FUNCTION_BLOCK "Jdrk_RS_WS_N01_8"   // FB31, SCL
{ S7_Optimized_Access := 'TRUE' }
VERSION : 0.1
   VAR_OUTPUT
      Temperature : Real;
   END_VAR
   VAR_IN_OUT
      mb_query : "mb_query";
   END_VAR
   VAR
      sb : "mb_station_block_udt";
   END_VAR
   VAR RETAIN
      offset : Real;
   END_VAR
   VAR_TEMP
      tmp : Int;
   END_VAR
BEGIN
   // JDRK - RS-WS-N01-8 - Temperature and Humidity sensor

   "mb_station_block_header"(sb := #sb, mb_query := #mb_query);

   #mb_query(mb_addr := 1,
             mode := #mb_query.c.read.input_reg,
             data_addr := 1,
             data_ptr := #tmp);

   IF #mb_query.Done THEN
       #Temperature := INT_TO_REAL(#tmp) / 10 + #offset;
   END_IF;

   "mb_station_block_footer"(sb := #sb, mb_query := #mb_query);
END_FUNCTION_BLOCK

FUNCTION_BLOCK "keller_pressure_transmitters"   // FB32, SCL
{ S7_Optimized_Access := 'TRUE' }
VERSION : 0.1
   VAR_INPUT
      mb_addr : USInt;
   END_VAR
   VAR_IN_OUT
      mb_query : "mb_query";
   END_VAR
   VAR
      sb : "mb_station_block_udt";
      data : Struct
         pressure_sensor_1 : Real;
         pressure_sensor_2 : Real;
         temperature : Real;
         temperature_sensor_1 : Real;
         temperature_sensor_2 : Real;
      END_STRUCT;
   END_VAR
BEGIN
   // Keller, Series 30 and Series 40 - Pressure transmitters
   // 
   // http://www.keller-druck.com/picts/pdf/engl/comm_protocol_e.pdf

   "mb_station_block_header"(sb := #sb,
                             mb_query := #mb_query);

   #mb_query(mb_addr := #mb_addr,
             mode := #mb_query.c.read.holding_reg,
             data_addr := 2,
             data_ptr := #data);

   "mb_station_block_footer"(sb := #sb,
                             mb_query := #mb_query);
END_FUNCTION_BLOCK

FUNCTION_BLOCK "Mjk_expert"   // FB35, SCL
{ S7_Optimized_Access := 'TRUE' }
VERSION : 0.1
   VAR_INPUT
      mb_addr : USInt;
   END_VAR
   VAR_IN_OUT
      mb_query : "mb_query";
   END_VAR
   VAR
      sb : "mb_station_block_udt";
      data : Struct
         CH0 : Real;   // calculated_value (User-specific)
         P1 : Real;   // Pressure sensor 1
         P2 : Real;   // Pressure sensor 2
         T : Real;   // Temperature
         T1 : Real;   // Temperature sensor 1
         T2 : Real;   // Temperature sensor 2
      END_STRUCT;
   END_VAR
BEGIN
   // MJK - Expert 700-7060-7070 - Pressure transmitters

   "mb_station_block_header"(sb := #sb,
                             mb_query := #mb_query);
   #mb_query.mb_addr := #mb_addr;

   #mb_query.mode := #mb_query.c.read.holding_reg;
   #mb_query(data_addr := 0,
             data_ptr := #data);

   "mb_station_block_footer"(sb := #sb,
                             mb_query := #mb_query);
END_FUNCTION_BLOCK

FUNCTION_BLOCK "Moxa_ioLogik_R1200"   // FB36, SCL
{ S7_Optimized_Access := 'TRUE' }
VERSION : 0.1
   VAR_INPUT
      mb_addr : UInt;
   END_VAR
   VAR_IN_OUT
      mb_query : "mb_query";
   END_VAR
   VAR
      sb : "mb_station_block_udt";
      in : Array[0..15] of Bool;
      out : Array[0..15] of Bool;
   END_VAR
BEGIN
   // Moxa - ioLogik R1200
   // 
   // Web: https://www.moxa.com/doc/man/ioLogik_R1200_Series_UM_e3.1.pdf

   "mb_station_block_header"(sb := #sb,
                             mb_query := #mb_query);
   #mb_query.mb_addr := #mb_addr;

   #mb_query(mode := #mb_query.c.read.discrete_input,
             data_addr := 0,
             data_ptr := #in);

   #mb_query(mode := #mb_query.c.write.discrete_output,
             data_addr := 16#140,
             data_ptr := #out);

   "mb_station_block_footer"(sb := #sb,
                             mb_query := #mb_query);
END_FUNCTION_BLOCK

FUNCTION_BLOCK "MTS_sensors_M_Series"   // FB37, SCL
{ S7_Optimized_Access := 'TRUE' }
VERSION : 0.1
   VAR_INPUT
      mb_addr : UInt;
   END_VAR
   VAR_OUTPUT
      level : Real;
      temperature : Real;
   END_VAR
   VAR_IN_OUT
      mb_query : "mb_query";
   END_VAR
   VAR
      sb : "mb_station_block_udt";
      query_1 : Struct
         product_level : DInt;
         Interface_level : DInt;
         roof_level : DInt;
         temperature : Array[1..5] of DInt;
         temperature_avg : DInt;
      END_STRUCT;
   END_VAR
BEGIN
   // MTS sensors - M-Series - Liquid-Level Sensors
   // Web: http://www.mtssensors.com/fileadmin/media/pdfs/550791.pdf

   "mb_station_block_header"(sb := #sb,
                             mb_query := #mb_query);
   #mb_query.mb_addr := #mb_addr;

   #mb_query.mode := #mb_query.c.mode.read;
   #mb_query(data_addr := 30001,
             data_ptr := #query_1);

   "mb_station_block_footer"(sb := #sb,
                             mb_query := #mb_query);

   #level := DINT_TO_REAL(#query_1.product_level) * 0.001;
   #temperature := DINT_TO_REAL(#query_1.temperature_avg) * 0.0001;
END_FUNCTION_BLOCK

FUNCTION_BLOCK "Novus_tht"   // FB38, SCL
{ S7_Optimized_Access := 'TRUE' }
VERSION : 0.1
   VAR_INPUT
      mb_addr : USInt;
   END_VAR
   VAR_OUTPUT
      temperature : Int;
      humidity : Int;
   END_VAR
   VAR_IN_OUT
      mb_query : "mb_query";
   END_VAR
   VAR
      sb : "mb_station_block_udt";
      serial_number : DWord;
      raw_values : Struct
         temp : Int;
         hum : Int;
      END_STRUCT;
   END_VAR
BEGIN
   // - Novus - RHT (Temperature transmitter)
   // - http://www.novusautomation.com/downloads/Arquivos/v10x_b_manual_rht_wm-dm-p10_485_lcd_%20english.pdf

   "mb_station_block_header"(sb := #sb, mb_query := #mb_query);
   #mb_query.mb_addr := #mb_addr;

   #mb_query.mode := #mb_query.c.read.holding_reg;
   #mb_query(data_addr := 7, data_ptr := #raw_values);
   #mb_query(data_addr := 0, data_ptr := #serial_number);

   "mb_station_block_footer"(sb := #sb, mb_query := #mb_query);

   #temperature := #raw_values.temp / 10;
   #humidity := #raw_values.hum / 10;
END_FUNCTION_BLOCK

FUNCTION_BLOCK "Onicon_F5100"   // FB39, SCL
{ S7_Optimized_Access := 'TRUE' }
VERSION : 0.1
   VAR_INPUT
      mb_addr : USInt;
   END_VAR
   VAR_IN_OUT
      mb_query : "mb_query";
   END_VAR
   VAR
      sb : "mb_station_block_udt";
      reset : Bool;
      query1 : Struct
         flow_total : UDInt;
      END_STRUCT;
      query2 : Struct
         flow_rate : Real;
         temperature : Real;
      END_STRUCT;
   END_VAR
BEGIN
   // Onicon - F-5100
   // http://www.onicon.com/pdfs/0669-7-F-5100-MOD-Network-Interface-Installation-Guide-09-15.pdf

   "mb_station_block_header"(sb := #sb,
                             mb_query := #mb_query);
   #mb_query.mb_addr := #mb_addr;

   #mb_query.data_addr := 312; // 313 - 1
   IF #reset THEN
       #query1.flow_total := 0;
       #mb_query(mode := #mb_query.c.write.holding_reg,
                 data_ptr := #query1.flow_total);
       IF #mb_query.stat.done THEN
           #reset := false;
       END_IF;
   ELSE
       #mb_query(mode := #mb_query.c.read.holding_reg,
                 data_ptr := #query1);
   END_IF;

   #mb_query(mode := #mb_query.c.read.holding_reg,
             data_addr := 578, // 579 - 1,
             data_ptr := #query2);

   "mb_station_block_footer"(sb := #sb,
                             mb_query := #mb_query);
END_FUNCTION_BLOCK

FUNCTION_BLOCK "Phoenix_Contact_UPS"   // FB40, SCL
{ S7_Optimized_Access := 'TRUE' }
VERSION : 0.1
   VAR_INPUT
      mb_addr : UInt;
   END_VAR
   VAR_IN_OUT
      mb_query : "mb_query";
   END_VAR
   VAR
      sb : "mb_station_block_udt";
      read1 : Struct
         remote : Word;
         BatteryMode : Word;
         ShutdownEvent : Word;
         BatteryCharging : Word;
      END_STRUCT;
      read2 : Struct
         OutputVoltage_mV : UInt;
      END_STRUCT;
      read3 : Struct
         SocStateOfCharge : UInt;   // [%]
         SocResidualBackupTimeM : UInt;   // Minute
      END_STRUCT;
      read4 : Struct
         BatteryVoltage_mV : UInt;
         BatteryTemperature : UInt;   // Kelvin
         OutputVoltage2_mV : UInt;
         SocResidualBackupTimeS : UInt;
         BatteryNomCapacityWs : UInt;
      END_STRUCT;
      read5 : Struct
         BatteryDischaCurrent : UInt;
         BatteryDetectedUnits : UInt;
         BatteryNomCapacitymAh : UInt;
         BatteryInstalledType : UInt;
      END_STRUCT;
      read6_Alarm : Struct
         x08 : Bool;
         x09_no_battery : Bool;
         x10_inconsistent_technology : Bool;
         x11_overload_cutoff : Bool;
         "x12_Low_battery_(Voltage)" : Bool;
         "x13_Low_battery_(Charge)" : Bool;
         "x14_Low_battery_(Time)" : Bool;
         x15 : Bool;
         "x00_End_of_life_(SOH)" : Bool;
         x01 : Bool;
         x02 : Bool;
         x03 : Bool;
         "x04_End_of_life_(Resitance)" : Bool;
         "x05_Endof_life_(Resitance)" : Bool;
         "x06_End_of_life_(Time)" : Bool;
         "x07_End_of_life_(Voltage)" : Bool;
      END_STRUCT;
   END_VAR
BEGIN
   // Phoenix Contact - UPS
   // QUINT UPS-IQ, TRIO-UPS
   // Web: https://media.digikey.com/pdf/Data%20Sheets/
   //      Phoenix%20Contact%20PDFs/2320461_Ds.pdf

   "mb_station_block_header"(sb := #sb, mb_query := #mb_query);
   #mb_query.mb_addr := #mb_addr;

   #mb_query.mode := #mb_query.c.read.holding_reg;
   #mb_query(data_addr := 29696, data_ptr := #read1);
   #mb_query(data_addr := 29745, data_ptr := #read2);
   #mb_query(data_addr := 29749, data_ptr := #read3);
   #mb_query(data_addr := 29792, data_ptr := #read4);
   #mb_query(data_addr := 29798, data_ptr := #read5);
   #mb_query(data_addr := 29840, data_ptr := #read6_Alarm);

   "mb_station_block_footer"(sb := #sb, mb_query := #mb_query);
END_FUNCTION_BLOCK

FUNCTION_BLOCK "Rotork_Mk_3_option_card"   // FB44, SCL
{ S7_Optimized_Access := 'TRUE' }
VERSION : 0.1
   VAR_INPUT
      mb_addr : UInt;
   END_VAR
   VAR_IN_OUT
      mb_query : "mb_query";
   END_VAR
   VAR
      sb : "mb_station_block_udt";
      read1 : Struct
         x00_actuator_moving : Bool;
         "x01_Close position limit" : Bool;
         "x02_Open position limit" : Bool;
         "x03_Valve running close" : Bool;
         "x04_Valve running open" : Bool;
         "x05_Selector in remote" : Bool;
         "x06_Selector in local stop" : Bool;
         "x07_Selector in local" : Bool;
         "x08_Thermostat tripped" : Bool;
         "x09_Monitor relay" : Bool;
         "x10_Valve obstructed" : Bool;
         "x11_Valve jammed" : Bool;
         "x12_Manual movement" : Bool;
         "x13_MIT_Interrupter timer" : Bool;
         "x14_Position control enabled" : Bool;
         "x15_Watchdog Recovery" : Bool;
         "x16_Battery low" : Bool;
         "x17_Open Interlock input active" : Bool;
         "x18_Close Interlock input active" : Bool;
         "x19_Hard wired input DI-1 (open)" : Bool;
         "x20_Hard wired input DI-2 (close)" : Bool;
         "x21_Hard wired input DI-3 (stop)" : Bool;
         "x22_Hard wired input DI-4 (ESD)" : Bool;
         x23 : Bool;
         x24 : Bool;
         x25 : Bool;
         "x26_Control contention" : Bool;
         "x27_Partial stroke test in progress" : Bool;
         "x28_Partial stroke test error" : Bool;
         "x29_General alarm" : Bool;
         x30 : Bool;
         x31 : Bool;
      END_STRUCT;
      read2 : Struct
         instantaneous_torque : Int;
         valve_position : Int;   // x10 %
         analogue_input : Int;
      END_STRUCT;
      write1 : Struct
         stop : Bool;
         close : Bool;
         open : Bool;
         emergency_shut_down : Bool;
         output_DO_1 : Bool;
         output_DO_2 : Bool;
         output_DO_3 : Bool;
         output_DO_4 : Bool;
      END_STRUCT;
      write2 : Struct
         actuator_digital_control : Bool;
         position_demand_output : Bool;
      END_STRUCT;
      actuator_tag_name : String[12];
      action_on_loss_of_comms : Int;
   END_VAR
BEGIN
   // Rotork  - Mk 3 Option Card

   // http://www.rotork.com/en/product/index/modbusliterature
   // Publication PUB091-004-00_0715

   "mb_station_block_header"(sb := #sb, mb_query := #mb_query);
   #mb_query.mb_addr := #mb_addr;

   #mb_query.mode := #mb_query.c.read.discrete_input;
   #mb_query(data_addr := 0, data_ptr := #read1);

   #mb_query.mode := #mb_query.c.read.holding_reg;
   #mb_query(data_addr := 2, data_ptr := #read2);
   #mb_query(data_addr := 26, data_ptr := #actuator_tag_name);

   #mb_query.mode := #mb_query.c.write.discrete_output;
   #mb_query(data_addr := 0, data_ptr := #write1);

   #mb_query.mode := #mb_query.c.write.holding_reg;
   // 0=No-Action, 1=Open, 3=Close, 5=Stop, 7=Position
   #mb_query(data_addr := 7, data_ptr := #action_on_loss_of_comms);
   #mb_query(data_addr := 5, data_ptr := #write2);

   "mb_station_block_footer"(sb := #sb, mb_query := #mb_query);
END_FUNCTION_BLOCK

FUNCTION_BLOCK "SensorsONE_DCT_531"   // FB52, SCL
{ S7_Optimized_Access := 'TRUE' }
VERSION : 0.1
   VAR_INPUT
      mb_addr : UInt;
   END_VAR
   VAR_IN_OUT
      mb_query : "mb_query";
   END_VAR
   VAR
      sb : "mb_station_block_udt";
      data : Struct
         serial_number : UDInt;
         date_last_calibration : UDInt;
         upper_range_pressure : Real;
         lower_range_pressure : Real;
         actual_pressure : Real;
         max_pressure : Real;
         min_pressure : Real;
         upper_range_temperature : Real;
         lower_range_temperature : Real;
         actual_temperature : Real;
         max_temperature : Real;
         min_temperature : Real;
      END_STRUCT;
   END_VAR
BEGIN
   // SensorsONE - DCT 531
   // 
   // https://www.sensorsone.com/dct-531-modbus-rtu-rs485-pressure-sensor/

   "mb_station_block_header"(sb := #sb,
                             mb_query := #mb_query);
   #mb_query.mb_addr := #mb_addr;

   #mb_query.mode := #mb_query.c.read.input_reg;
   #mb_query(data_addr := 0,
             data_ptr := #data);

   "mb_station_block_footer"(sb := #sb,
                             mb_query := #mb_query);
END_FUNCTION_BLOCK

FUNCTION_BLOCK "Sierra_thermal_mass_flow_meters"   // FB61, SCL
{ S7_Optimized_Access := 'TRUE' }
VERSION : 0.1
   VAR_INPUT
      mb_addr : UInt;
      reset_totalizer : Bool := 1;
   END_VAR
   VAR_IN_OUT
      mb_query : "mb_query";
   END_VAR
   VAR
      sb : "mb_station_block_udt";
      data : Struct
         flow : Real;
         totalizer : DInt;
      END_STRUCT;
      serial_number : String[12];
   END_VAR
   VAR_TEMP
      "int" : Int;
   END_VAR
BEGIN
   // Sierra - 600/700 Series - Thermal mass flow meters
   // Models: 620S, 620S-BT, 640S, 760S, 780S, and 780S-UHP

   // Web: https://www.ccontrols.com/support/dp/600-700-modbus-instruction-manual.pdf

   "mb_station_block_header"(sb := #sb,
                             mb_query := #mb_query);
   #mb_query.mb_addr := #mb_addr;

   #mb_query.mode := #mb_query.c.mode.read;
   #mb_query(data_addr := 40001,
             data_ptr := #data);
   #mb_query(data_addr := 40016,
             data_ptr := #serial_number);

   IF #reset_totalizer THEN
       #mb_query.mode := #mb_query.c.mode.write;
       #"int" := 1;
       #mb_query(data_addr := 40008,
                 data_ptr := #"int");
   END_IF;

   "mb_station_block_footer"(sb := #sb,
                             mb_query := #mb_query);
END_FUNCTION_BLOCK

FUNCTION_BLOCK "Smart_biene_sb_hl"   // FB62, SCL
{ S7_Optimized_Access := 'TRUE' }
VERSION : 0.1
   VAR_INPUT
      mb_addr : UInt;
   END_VAR
   VAR_IN_OUT
      mb_query : "mb_query";
   END_VAR
   VAR
      s : "mb_station_block_udt";
      data : Struct
         "Min measuring range" : Word;
         "Max measuring range" : Word;
         "Pressure Value" : Word;
         "High Pressure" : Word;
         "Low Pressure" : Word;
         stat : Word;
         model : String[12];
         serial : String[12];
         unit : Int;
      END_STRUCT;
      "a" : Struct
         x08 : Bool;
         x09 : Bool;
         x10 : Bool;
         x11 : Bool;
         x12 : Bool;
         x13 : Bool;
         x14 : Bool;
         x15 : Bool;
         x00 : Bool;
         x01 : Bool;
         x02 : Bool;
         x03 : Bool;
         x04 : Bool;
         x05 : Bool;
         x06 : Bool;
         x07 : Bool;
      END_STRUCT;
   END_VAR
BEGIN
   // Smart Biene - SB-HL - Hydrostatic Level Transmitter
   // 
   // Web: http://smartbiene.com/images/pdf/hydrostatic-level/
   //      Hydrostatic%20level-SP-HL-01-ModbusRTU.pdf

   "mb_station_block_header"(sb := #s,
                             mb_query := #mb_query);
   #mb_query.mb_addr := #mb_addr;

   #mb_query.mode := #mb_query.c.read.holding_reg;
   #mb_query(data_addr := 0,
             data_ptr := #data);

   "mb_station_block_footer"(sb := #s,
                             mb_query := #mb_query);

   (*
   Unit:
   0-mbar
   1-bar
   2-PSI
   3-KPa
   4-MPa
   5-Kg/cm2
   6-mmHg
   7-mmH2O
   8-inHg
   9-inH2O 
   *)
END_FUNCTION_BLOCK

FUNCTION_BLOCK "Socomec_diris"   // FB63, SCL
{ S7_Optimized_Access := 'TRUE' }
VERSION : 0.1
   VAR_INPUT
      mb_addr : USInt;
      old_mapping : Bool;
   END_VAR
   VAR_OUTPUT
      data : Struct
         voltage_L_L : Array[1..3] of Real;   // 1->L1-L2, 2->L2-L3, 3->L3-L1
         voltage_L_N : Array[1..3] of Real;
         frequency : Real;
         current : Array[1..3] of Real;
         neutral_current : Real;
         sum_active_power : Real;
         sum_reactive_power : Real;
         sum_apparent_power : Real;
         sum_power_factor : Real;   // -: leading and + : lagging
         power_active : Array[1..3] of Real;
         power_reactive : Array[1..3] of Real;
         power_apparent : Array[1..3] of Real;
         power_factor : Array[1..3] of Real;
      END_STRUCT;
   END_VAR
   VAR_IN_OUT
      mb_query : "mb_query";
   END_VAR
   VAR
      sb : "mb_station_block_udt";
      query_1 : Struct
         voltage_L_L : Array[1..3] of DInt;   // 1->L1-L2, 2->L2-L3, 3->L3-L1
         voltage_L_N : Array[1..3] of DInt;
         frequency : DInt;
         current : Array[1..3] of DInt;
         neutral_current : DInt;
         sum_active_power : DInt;
         sum_reactive_power : DInt;
         sum_apparent_power : DInt;
         sum_power_factor : DInt;   // -: leading and + : lagging
         power_active : Array[1..3] of DInt;
         power_reactive : Array[1..3] of DInt;
         power_apparent : Array[1..3] of DInt;
         power_factor : Array[1..3] of DInt;
      END_STRUCT;
      query_2_temperature : DInt;
   END_VAR
   VAR_TEMP
      j : Int;
   END_VAR
BEGIN
   // Socomec Diris A40/A41 - Power meter
   // https://www.socomec.com/files/live/sites/systemsite/files/SCP/
   // 6_gestion_energie/diris/diris_a40/536181B_GB_Ethernet.pdf

   // old_mapping:
   // http://www.ferrazshawmutsales.com/pdfs/cdr_27038_RS485_JBus-ModBus.pdf

   "mb_station_block_header"(sb := #sb,
                             mb_query := #mb_query);
   #mb_query.mb_addr := #mb_addr;

   #mb_query.mode := #mb_query.c.read.holding_reg;

   #mb_query(data_addr := SEL(G := #old_mapping, IN0 := 50514, IN1 := 768),
             data_ptr := #query_1);

   IF NOT #old_mapping THEN
       #mb_query(data_addr := 51457,
                 data_ptr := #query_2_temperature);
   END_IF;

   "mb_station_block_footer"(sb := #sb,
                             mb_query := #mb_query);

   (* IF #s.out.error_comm THEN
       FOR #j := 1 TO 3 DO
           #query_1.voltage_L_L[#j] := 0;
           #query_1.voltage_L_N[#j] := 0;
           #query_1.current[#j] := 0;
           #query_1.power_active[#j] := 0;
           #query_1.power_reactive[#j] := 0;
           #query_1.power_apparent[#j] := 0;
           #query_1.power_factor[#j] := 0;
       END_FOR;
       #query_1.frequency := 0;
       #query_1.neutral_current := 0;
       #query_1.sum_active_power := 0;
       #query_1.sum_reactive_power := 0;
       #query_1.sum_apparent_power := 0;
       #query_1.sum_power_factor := 0;

       #query_2_temperature := 0;
   END_IF; // *)

   FOR #j := 1 TO 3 DO
       #data.voltage_L_L[#j] := DINT_TO_REAL(#query_1.voltage_L_L[#j]) / 100;
       #data.voltage_L_N[#j] := DINT_TO_REAL(#query_1.voltage_L_N[#j]) / 100;
       #data.current[#j] := DINT_TO_REAL(#query_1.current[#j]) / 1000;
       #data.power_active[#j] := DINT_TO_REAL(#query_1.power_active[#j]) / 100;
       #data.power_reactive[#j] := DINT_TO_REAL(#query_1.power_reactive[#j]) / 100;
       #data.power_apparent[#j] := DINT_TO_REAL(#query_1.power_apparent[#j]) / 100;
       #data.power_factor[#j] := DINT_TO_REAL(#query_1.power_factor[#j]) / 1000;
   END_FOR;
   #data.frequency := DINT_TO_REAL(#query_1.frequency) / 100;
   #data.neutral_current := DINT_TO_REAL(#query_1.neutral_current) / 100;
   #data.sum_active_power := DINT_TO_REAL(#query_1.sum_active_power) / 100;
   #data.sum_reactive_power := DINT_TO_REAL(#query_1.sum_reactive_power) / 100;
   #data.sum_apparent_power := DINT_TO_REAL(#query_1.sum_apparent_power) / 100;
   #data.sum_power_factor := DINT_TO_REAL(#query_1.sum_power_factor) / 1000;
END_FUNCTION_BLOCK

FUNCTION_BLOCK "Sparling_Instruments_Tiger_Mag"   // FB64, SCL
{ S7_Optimized_Access := 'TRUE' }
VERSION : 0.1
   VAR_INPUT
      mb_addr : USInt;
   END_VAR
   VAR_IN_OUT
      mb_query : "mb_query";
   END_VAR
   VAR
      sb : "mb_station_block_udt";
      read1 : Struct
         flow : Real;   // 0.01 [Hz]
         total_fwd : UDInt;   // 0.1 [A]
         total_rev : UDInt;
         unit_flow : String[4];
         unit_total : String[4];
         total_registration : Real;
      END_STRUCT;
      serial_number : UDInt;
   END_VAR
BEGIN
   // Sparling Instruments - Tiger Mag 
   // FM656, FM657, FM626, FM627, FM626 Sanitary
   // http://www.sparlinginstruments.com/documents/IDS-TMEP-160323.PDF
   // Revision 160323

   "mb_station_block_header"(sb := #sb,
                             mb_query := #mb_query);
   #mb_query.mb_addr := #mb_addr;

   #mb_query.mode := #mb_query.c.mode.read;
   #mb_query(data_addr := 30001,
             data_ptr := #read1);
   #mb_query(data_addr := 31003,
             data_ptr := #serial_number);

   "mb_station_block_footer"(sb := #sb,
                             mb_query := #mb_query);

   (*
   Terminal RS-485 Bus:
   1-RX  -> A+
   2-TX  -> B-
   3-GND -> GND
   4-DTR -> N/A Not used

   Default comm. param:
   19200 bps, even parity. 
    Slave ID: 1.
   *)
END_FUNCTION_BLOCK

FUNCTION_BLOCK "Syxthsense_TEHR_M"   // FB70, SCL
TITLE = Syxthsense - TEHR-M - Temperature transmitter
{ S7_Optimized_Access := 'TRUE' }
AUTHOR : OlaBjornli
VERSION : 0.1
   VAR_INPUT
      mb_addr : USInt := 1;
   END_VAR
   VAR_OUTPUT
      temperature : Real;   // [Â°C]
      analogue_output : Real;   // [Â°F]
      potentiometer_position : Real;   // [%]
   END_VAR
   VAR_IN_OUT
      mb_query : "mb_query";
   END_VAR
   VAR
      sb : "mb_station_block_udt";
      read1 : Struct
         temperature : Int;   // [Â°C]
         analogue_output : Int;   // [Â°F]
         potentiometer_position : Int;   // [%]
      END_STRUCT;
   END_VAR
BEGIN
   // http://www.syxthsense.com/product/product_pdf/SN1.174-TEHR-M.pdf

   "mb_station_block_header"(sb := #sb, mb_query := #mb_query);

   #mb_query(mb_addr := #mb_addr,
             mode := #mb_query.c.mode.read,
             data_addr := 30001,
             data_ptr := #read1);
   #temperature := INT_TO_REAL(#read1.temperature) / 10;
   #analogue_output := INT_TO_REAL(#read1.analogue_output) / 10;
   #potentiometer_position := INT_TO_REAL(#read1.potentiometer_position) / 10;

   "mb_station_block_footer"(sb := #sb, mb_query := #mb_query);
END_FUNCTION_BLOCK

FUNCTION_BLOCK "Telemecanique_Schneider_Altivar_21_inverter"   // FB71, SCL
{ S7_Optimized_Access := 'TRUE' }
VERSION : 0.1
   VAR_INPUT
      mb_addr : UInt;
      ref : Real;
   END_VAR
   VAR_IN_OUT
      mb_query : "mb_query";
   END_VAR
   VAR
      sb : "mb_station_block_udt";
      read1 : Struct
         "Output frequency" : Word;
         stat : Struct
            x08 : Bool;
            x09_Reverse : Bool;
            x10_Run : Bool;
            x11_Coast_stop : Bool;
            x12_Emergency_stop : Bool;
            x13_Standby_ST_ON : Bool;   // Standby: Initialization completed, not failure stop status, not alarm stop status (MOFF, LL forced stop or forced stop due to a momentary power failure), ST=ON, and RUN=ON
            x14_Standby : Bool;   // Standby: Initialization completed, not failure stop status, and not alarm stop status (MOFF, LL forced stop or forced stop due to a momentary power failure)
            x15_Local : Bool;
            x00_Failure_FL : Bool;
            x01_Failure : Bool;
            x02_Alarm : Bool;
            x03_Main_circuit_undervoltage : Bool;
            x04_THR_2 : Bool;   // THR1: PT=set value, vL, vb, Thr - THR2: PT=0, F170, F172, F173
            x05_PI_control_OFF : Bool;
            x06_Acceleration2_deceleration2 : Bool;
            x07_DC_braking : Bool;
         END_STRUCT;
      END_STRUCT;
      read2 : Struct
         Command_mode : Int;   // 0:Terminal board, 1:Operation panel, 2:Serial
         "Setpoint mode" : Int;   // 1 VIA, 2 VIB, 3 Operation panel, 4 Serial, 5 TB up down frequency, 255 Preset speed operation
      END_STRUCT;
      read3_alarm : Struct
         x08_Over_torque : Bool;
         x09_Cumulative_operation_hours : Bool;
         x10 : Bool;
         x11 : Bool;
         x12 : Bool;
         "x13_Main circuit_undervoltage" : Bool;   // same as MS-relay status
         x14_Decelerating_stopping : Bool;   // Related: F256 setting. At the time of the instant blackout, Forced deceleration/stop
         x15_Decelerating_stopping : Bool;   // Related: F302 setting. An automatic stop during the lower limit frequency continuance
         x00_Overcurrent : Bool;
         x01_Inverter_overload : Bool;
         x02_Motor_overload : Bool;
         x03_Overheat : Bool;
         x04_Overvoltage : Bool;
         x05_Main_circuit_undervoltage : Bool;
         x06 : Bool;
         x07_Undercurrent : Bool;
      END_STRUCT;
      read4_alarm2 : Struct
         x08 : Bool;
         x09 : Bool;
         x10 : Bool;
         x11 : Bool;
         x12 : Bool;
         x13 : Bool;
         x14 : Bool;
         x15 : Bool;
         x00_Fan_life_alarm : Bool;
         x01_Circuit_board_life : Bool;
         x02_Main_circuit_capacitor_life : Bool;
         x03_User_set_alarm : Bool;
         x04 : Bool;
         x05 : Bool;
         x06 : Bool;
         x07 : Bool;
      END_STRUCT;
      read5_trip_code : UInt;
      write1 : Struct
         cmd : Struct
            x08 : Bool;
            x09_Reverse : Bool;
            x10_Run : Bool;
            x11_Coast_stop : Bool;
            x12_Emergency_stop : Bool;
            x13_Fault_reset : Bool;
            x14_Setpoint_priority : Bool;   // Enabled regardless of the setting of FMOD
            x15_Command_priority : Bool;   // Enabled regardless of the setting of CMOD
            x00_Preset_speed_b0 : Bool := TRUE;
            x01_Preset_speed_b1 : Bool;
            x02_Preset_speed_b2 : Bool;
            x03 : Bool;
            x04_thr2 : Bool;   // THR1 : PT=set value, vL, vb, tHr - THR2 : PT=0, F170, F172, F173
            x05_PI_control : Bool;   // 0:Normal operation, 1:PI OFF
            x06_Acceleration_deceleration_pattern_2 : Bool;   // 0: Acceleration deceleration pattern 1
            x07_DC_braking : Bool;
         END_STRUCT;
         ref : UInt;
      END_STRUCT;
   END_VAR
BEGIN
   // Telemecanique (Schneider) - Altivar 21 inverter
   // VFD (AC-drive)
   // http://www2.schneider-electric.com/resources/sites/SCHNEIDER_ELECTRIC/
   // content/live/FAQS/12000/FA12122/en_US/Altivar%2021%20Modbus%20manual.pdf

   "mb_station_block_header"(sb := #sb, mb_query := #mb_query);
   #mb_query.mb_addr := #mb_addr;

   #mb_query.mode := #mb_query.c.read.holding_reg;
   #mb_query(data_addr := 16#fd00, data_ptr := #read1);
   #mb_query(data_addr := 16#fe45, data_ptr := #read2);
   #mb_query(data_addr := 16#fe91, data_ptr := #read3_alarm);
   #mb_query(data_addr := 16#fe79, data_ptr := #read4_alarm2);
   #mb_query(data_addr := 16#FC90, data_ptr := #read5_trip_code);

   #write1.ref := REAL_TO_UINT(#ref * 100);
   #write1.cmd.x10_Run := #ref <> 0;
   #mb_query.mode := #mb_query.c.write.holding_reg;
   #mb_query(data_addr := 16#fa00, data_ptr := #write1);

   "mb_station_block_footer"(sb := #sb, mb_query := #mb_query);

   (* Trip code
   NErr     0  0  No error
   OC1      1  1  Over-current during acceleration
   OC2      2  2  Over-current during deceleration
   OC3      3  3  Over-current during constant speed operation
   OCL      4  4  Over-current in load at startup
   OCA      5  5  Short circuit in arm
   EPHI     8  8  Input phase failure
   EPHO     9  9  Output phase failure
   OP1      A 10 Overvoltage during acceleration
   OP2      B 11 Overvoltage during deceleration
   OP3      C 12 Overvoltage during constant speed operation
   OL1      D 13 Over-LOAD in inverter
   OL2      E 14 Over-LOAD in motor
   OH      10 16 Overheat trip
   E       11 17 Emergency stop
   EEP1    12 18 EEPROM fault 1 (writing error)
   EEP2    13 19 EEPROM fault 2 (reading error)
   EEP3    14 20 EEPROM fault 3 (internal fault)
   Err2    15 21 RAM fault
   Err3    16 22 ROM fault
   Err4    17 23 CPU fault
   Err5    18 24 Communication error trip
   Err7    1A 26 Current detector fault
   Err8    1B 27 Optional circuit board type error
   UC      1D 29 Small-current trip
   UP1     1E 30 Trip due to undervoltage in main circuit
   Ot      20 32 Over-torque trip
   EF2     22 34 Ground fault trip (hardware detection)
   OC1P    25 37 Overcurrent flowing in element during acceleration
   OC2P    26 38 Overcurrent flowing in element during deceleration
   OC3P    27 39 Overcurrent flowing in element during operation
   EtYP    29 41 Inverter type error
   OH2     2E 46 External thermal input
   SOUt    2F 47 VIA cable break
   E-18    32 50 Break in an analog signal cable
   E-19    33 51 CPU fault
   E-20    34 52 Excess torque boost
   E-21    35 53 CPU fault
   Etn1    54 84 Auto-tuning error
   *)
END_FUNCTION_BLOCK

FUNCTION_BLOCK "Vacon_OPTC2_C8"   // FB72, SCL
{ S7_Optimized_Access := 'TRUE' }
VERSION : 0.1
   VAR_INPUT
      mb_addr : UInt;
      ref : Real;
   END_VAR
   VAR_OUTPUT
      actual_speed : Real;
      Output_Frequency : Real;   // hz
      Motor_Speed : Real;   // rpm
      Motor_Current : Real;   // A
      Motor_Torque : Real;   // %
      Motor_Power : Real;   // %
      Motor_Voltage : Real;   // V
      DC_link_voltage : Real;   // V
   END_VAR
   VAR_IN_OUT
      mb_query : "mb_query";
   END_VAR
   VAR
      sb : "mb_station_block_udt";
      write : Struct
         ctw : Struct
            byte0 : Bool;
            x00_run : Bool;
            x01_reverse : Bool;
            x02_reset : Bool;
            x03 : Bool;
            x04 : Bool;
            x05 : Bool;
            x06 : Bool;
            x07 : Bool;
         END_STRUCT;
         "General Control Word" : Word;
         speed_reference : Int;
      END_STRUCT;
      read : Struct
         status : Struct
            x08_TC_Speed_Limit_Not_Active : Bool;
            x09_Detected_Encoder_Direction_Counterclockwise : Bool;
            x10_UV_Fast_Stop_Not_Active : Bool;
            x11 : Bool;
            x12 : Bool;
            x13 : Bool;
            x14 : Bool;
            x15 : Bool;
            x00_ready : Bool;
            x01_RUN : Bool;
            x02_reverse : Bool;
            x03_Faulted : Bool;
            x04_Warning : Bool;
            x05_Ref_Frequency_reached : Bool;
            x06_Motor_is_running_at_zero_speed : Bool;
            x07_Flux_Ready : Bool;
         END_STRUCT;
         general_status : Struct
            x08 : Bool;
            x09 : Bool;
            x10 : Bool;
            x11 : Bool;
            x12 : Bool;
            x13_Fieldbus_control : Bool;
            "x14_Panel control" : Bool;
            x15_IO_control : Bool;
            x00 : Bool;
            x01 : Bool;
            x02 : Bool;
            x03 : Bool;
            x04 : Bool;
            x05 : Bool;
            x06 : Bool;
            x07 : Bool;
         END_STRUCT;
         actual_speed : Int;
         Output_Frequency : Int;   // 0.01 Hz
         Motor_Speed : Int;   // 1 rpm
         Motor_Current : Int;   // 0.1 A
         Motor_Torque : Int;   // 0.1 %
         Motor_Power : Int;   // 0.1 %
         Motor_Voltage : Int;   // 0.1 V
         DC_link_voltage : Int;   // 1 V
         Active_Fault_Code : Int;
      END_STRUCT;
   END_VAR
BEGIN
   // Vacon NX - OPTC2/C8 - AC drives
   // Modbus/N2 option board
   // Document code: DPD00899A , Date 19.01.2012
   // Web: http://www.vacon.com/ImageVaultFiles/id_3118/cf_2/
   //      Vacon-NX-OPTC2-C8-Modbus-N2-Board-User-Manual-DPD0.
   //      PDF?635223804391930000

   "mb_station_block_header"(sb := #sb, mb_query := #mb_query);
   #mb_query.mb_addr := #mb_addr;

   #mb_query.mode := #mb_query.c.read.holding_reg;

   #mb_query(data_addr := 42101, data_ptr := #read);
   #actual_speed := INT_TO_REAL(#read.actual_speed);
   #Output_Frequency := INT_TO_REAL(#read.Output_Frequency) * 0.01;
   #Motor_Speed := INT_TO_REAL(#read.Motor_Speed);
   #Motor_Current := INT_TO_REAL(#read.Motor_Current) * 0.1;
   #Motor_Torque := INT_TO_REAL(#read.Motor_Torque) * 0.1;
   #Motor_Power := INT_TO_REAL(#read.Motor_Power) * 0.1;
   #Motor_Voltage := INT_TO_REAL(#read.Motor_Voltage) * 0.1;
   #DC_link_voltage := INT_TO_REAL(#read.DC_link_voltage);

   // -------------------------------------------------------
   #mb_query.mode := #mb_query.c.write.holding_reg;

   #write.ctw.x00_run := #ref <> 0;
   #mb_query(data_addr := 42001, data_ptr := #write.ctw);
   #write.speed_reference := REAL_TO_INT(#ref * 100);
   #mb_query(data_addr := 42003, data_ptr := #write.speed_reference);

   "mb_station_block_footer"(sb := #sb, mb_query := #mb_query);
END_FUNCTION_BLOCK

FUNCTION_BLOCK "vega_vegabar_81"   // FB73, SCL
{ S7_Optimized_Access := 'TRUE' }
VERSION : 0.1
   VAR_INPUT
      mb_addr : UInt;
   END_VAR
   VAR_IN_OUT
      mb_query : "mb_query";
   END_VAR
   VAR
      sb : "mb_station_block_udt";
      read1 : Struct
         status : Struct
            x08 : Bool;
            x09 : Bool;
            x10 : Bool;
            x11 : Bool;
            x12 : Bool;
            x13 : Bool;
            x14 : Bool;
            x15 : Bool;
            x00_invalid_measurement_1 : Bool;
            x01_invalid_measurement_2 : Bool;
            x02_invalid_measurement_3 : Bool;
            x03_invalid_measurement_4 : Bool;
            x04 : Bool;
            x05 : Bool;
            x06 : Bool;
            x07 : Bool;
         END_STRUCT;
         z : Word;
         data : Array[1..4] of Real;
      END_STRUCT;
   END_VAR
BEGIN
   // Vega - VEGABAR 81

   "mb_station_block_header"(sb := #sb, mb_query := #mb_query);
   #mb_query.mb_addr := #mb_addr;

   #mb_query(mode := #mb_query.c.read.holding_reg,
             data_addr := 2000,
             data_ptr := #read1);

   "mb_station_block_footer"(sb := #sb, mb_query := #mb_query);

   (*
   Unit Code Measurement Unit:
   32 Degree Celsius
   33 Degree Fahrenheit
   40 US Gallon
   41 Liters
   42 Imperial Gallons
   43 Cubic Meters
   44 Feet
   45 Meters
   46 Barrels
   47 Inches
   48 Centimeters
   49 Millimeters
   111 Cubic Yards
   112 Cubic Feet
   113 Cubic Inches
   *)
END_FUNCTION_BLOCK

FUNCTION_BLOCK "Weg_CFW100"   // FB74, SCL
{ S7_Optimized_Access := 'TRUE' }
VERSION : 0.1
   VAR_INPUT
      mb_addr : UInt;
   END_VAR
   VAR_IN_OUT
      mb_query : "mb_query";
   END_VAR
   VAR
      sb : "mb_station_block_udt";
      r1 : Struct
         Output_Speed : UInt;   // 2
         Motor_Current : UInt;
         DC_Link_Voltage : UInt;
         Output_Frequency : UInt;
         Inverter_Status : UInt;
         Output_Voltage : UInt;
         Motor_Torque : UInt;
         Active_Current : UInt;
         digital_input : UInt;
      END_STRUCT;
      r2_staus : Struct
         x08_running : Bool;
         x09_ready : Bool;
         x10_forward : Bool;
         x11_jog_active : Bool;
         x12_remote_mode : Bool;
         x13_undervoltage : Bool;
         x14_ : Bool;
         x15_fault : Bool;
         x00 : Bool;
         x01 : Bool;
         x02 : Bool;
         x03 : Bool;
         x04 : Bool;
         x05_2nd_Ramp : Bool;   // 0: 1st Acceleration and deceleration ramp by P100 and P101.
         x06_configuration_state : Bool;
         x07_alarm : Bool;
         "a" : Struct
            x08 : Bool;
            x09 : Bool;
            x10 : Bool;
            x11 : Bool;
            x12 : Bool;
            x13 : Bool;
            x14 : Bool;
            x15 : Bool;
            x00 : Bool;
            x01 : Bool;
            x02 : Bool;
            x03 : Bool;
            x04 : Bool;
            x05 : Bool;
            x06 : Bool;
            x07 : Bool;
         END_STRUCT;
      END_STRUCT;
      _ : Bool;
      w1 : Struct
         Minimum_Frequency : UInt;
         Maximum_Frequency : UInt := 50;
         Maximum_Output_Current : UInt := 100;
      END_STRUCT;
      w2 : Struct
         "Acceleration Time" : UInt := 5;
         "Deceleration Time" : UInt := 10;
      END_STRUCT;
      w3_sel_rem : UInt := 1;   // 1 = Always Remote
      w4_Ref_sel : UInt := 9;   // 9=serial
      w5 : Struct
         controll_word : Struct
            x08 : Bool;
            x09 : Bool;
            x10 : Bool;
            x11 : Bool;
            x12 : Bool;
            x13 : Bool;
            x14 : Bool;
            x15 : Bool;
            x00_no_ramp_stop : Bool := TRUE;
            x01_start : Bool := TRUE;
            x02_Forward : Bool;
            x03_jog : Bool;
            x04_Remote : Bool := TRUE;
            "x05_2nd Ramp" : Bool;
            x06 : Bool;
            x07_Fault_Reset : Bool;
            "a" : Struct
               x08 : Bool;
               x09 : Bool;
               x10 : Bool;
               x11 : Bool;
               x12 : Bool;
               x13 : Bool;
               x14 : Bool;
               x15 : Bool;
               x00 : Bool;
               x01 : Bool;
               x02 : Bool;
               x03 : Bool;
               x04 : Bool;
               x05 : Bool;
               x06 : Bool;
               x07 : Bool;
            END_STRUCT;
         END_STRUCT;
         speed_ref : Int;
      END_STRUCT;
      w6_stop_mode : Int;
      w7_no_comm_action : Int := 1;   // 1 = Ramp Stop
      c : Int := 1;
      setup_finished : Bool;
   END_VAR
BEGIN
   // Weg - CFW100
   // 
   // Web: http://www.clrwtr.com/PDF/WEG/WEG-CFW100-Programming.pdf

   "mb_station_block_header"(sb := #sb,
                             mb_query := #mb_query);
   #mb_query.mb_addr := #mb_addr;

   #mb_query.mode := #mb_query.c.read.holding_reg;
   #mb_query(data_addr := 2,
             data_ptr := #r1);
   #mb_query(data_addr := 680,
             data_ptr := #r2_staus);

   #mb_query.mode := #mb_query.c.write.holding_reg;
   #mb_query(data_addr := 682,
             data_ptr := #w5);
   CASE #c OF
       1:
           #mb_query(data_addr := 133,
                     data_ptr := #w1);
       2:
           #mb_query(data_addr := 101,
                     data_ptr := #w2);
       3:
           #mb_query(data_addr := 220,
                     data_ptr := #w3_sel_rem);
       4:
           #mb_query(data_addr := 222,
                     data_ptr := #w4_Ref_sel);
       5:
           #mb_query(data_addr := 229,
                     data_ptr := #w6_stop_mode);
       6:
           #mb_query(data_addr := 313,
                     data_ptr := #w7_no_comm_action);
       ELSE:
           #c := 0;
   END_CASE;
   #c += BOOL_TO_INT(#mb_query.Done);

   "mb_station_block_footer"(sb := #sb,
                             mb_query := #mb_query);
   IF #sb.out.error_comm THEN
       #setup_finished := false;
   END_IF;

   (*
   P229 Stop mode:
   0 The inverter will apply the stop ramp programmed in P101 or P103.
   1 The motor will run free until it stops

   P006 Inverter Status:
   0 = Ready
   1 = Run
   2 = Undervoltage
   3 = Fault
   4 = Not Used
   5 = Configuration

   *)
END_FUNCTION_BLOCK

FUNCTION_BLOCK "Wika_GDT20_GDHT20"   // FB75, SCL
{ S7_Optimized_Access := 'TRUE' }
VERSION : 0.1
   VAR_INPUT
      mb_addr : UInt;
   END_VAR
   VAR_IN_OUT
      mb_query : "mb_query";
   END_VAR
   VAR
      sb : "mb_station_block_udt";
      data : Struct
         pressure_bar : Real;
         pressure_MPa : Real;
         pressure_Pa : Real;
         pressure_kPa : Real;
         pressure_psi : Real;
         pressure_N_cmÂ² : Real;
         Temperature_C : Real;
         Temperature_K : Real;
         Temperature_F : Real;
         gas_density_g_l : Real;
         gas_density_kg_m3 : Real;
         "Pressure_standardised_to 20_C" : Real;
         Humidity_Atmosphere_frost_point : Real;
         Humidity_Atmosphere_dew_point : Real;
         Humidity_Tank_pressure_frost_point : Real;
         Humidity_Tank_pressure_dew_point_1 : Real;
      END_STRUCT;
      tag : String[16];
      alarm : Struct
         x08_Failure_humidity_sensor : Bool;   // (only model GDHT-20)
         x09_Communication_error_humidity_sensor : Bool;   // (only model GDHT-20)
         x10_Re_occurring_Modbus_communication_error : Bool;   // Re-occurring ModbusÂ® communication error
         x11 : Bool;
         x12 : Bool;
         x13 : Bool;
         x14 : Bool;
         x15 : Bool;
         x00_Pressure_below_lower_limit : Bool;   // Pressure signal below the lower limit value (< 0 bar)
         x01_Pressure_above_upper_limit : Bool;
         x02_Pressure_sensor_failure : Bool;
         x03_Temperature_below_lower_limit : Bool;   // Temperature signal below the lower limit value (< -40 Â°C)
         x04_Temperature_above_upper_limit : Bool;
         x05_Communication_error_pressure_temperature_sensor : Bool;
         x06_Pressure_density_below_lower_limit : Bool;   // Pressure density below the lower limit value (liquefaction of SF6 gas)
         x07_Gas_density_above_upper_limit : Bool;   // Gas density above the upper limit value (> 80 g/l)
      END_STRUCT;
      reset_alarm : Bool;
   END_VAR
   VAR_TEMP
      "int" : Int;
   END_VAR
BEGIN
   // Wika - GDT-20, GDHT-20 (GDT-20, GDHT-20)
   // Pressure / temperature / Gas density / Humidity 
   // 
   // http://en-co.wika.de/upload/OI_GDT_GDHT_20_en_de_67032.pdf

   "mb_station_block_header"(sb := #sb,
                             mb_query := #mb_query);
   #mb_query.mb_addr := #mb_addr;

   #mb_query.mode := #mb_query.c.read.holding_reg;
   #mb_query(data_addr := 0,
             data_ptr := #data);
   #mb_query(data_addr := 113,
             data_ptr := #tag);
   #mb_query(data_addr := 200,
             data_ptr := #alarm);

   IF #reset_alarm THEN
       #"int" := 1;
       #mb_query(mode := #mb_query.c.write.holding_reg,
                 data_addr := 201,
                 data_ptr := #"int");
       IF #mb_query.Done THEN
           #reset_alarm := false;
       END_IF;
   END_IF;

   "mb_station_block_footer"(sb := #sb,
                             mb_query := #mb_query);


   (*
   Circular connector M12 x 1 (5-pin):
   1 C Reference potential RS-485 common
   2 UB Voltage supply (DC 17 ... 30 V)
   3 GND Ground
   4 A Signal RS-485
   5 B Signal RS-485
   *)
END_FUNCTION_BLOCK

FUNCTION_BLOCK "Yaskawa_e7_drive"   // FB76, SCL
{ S7_Optimized_Access := 'TRUE' }
VERSION : 0.1
   VAR_INPUT
      mb_addr : UInt;
   END_VAR
   VAR_IN_OUT
      mb_query : "mb_query";
   END_VAR
   VAR
      sb : "mb_station_block_udt";
      read1 : Struct
         stat : Struct
            x08 : Bool;
            x09 : Bool;
            x10 : Bool;
            x11 : Bool;
            x12 : Bool;
            x13 : Bool;
            x14 : Bool;
            x15 : Bool;
            x00_run : Bool;
            x01 : Bool;
            x02 : Bool;
            x03_reset_signal : Bool;
            x04_speed_agree : Bool;
            x05_inverter_ready : Bool;
            x06_minor_fault : Bool;
            x07_major_fault : Bool;
            "a" : Struct
               x08 : Bool;
               x09 : Bool;
               x10 : Bool;
               x11 : Bool;
               x12 : Bool;
               x13 : Bool;
               x14 : Bool;
               x15 : Bool;
               x00 : Bool;
               x01 : Bool;
               x02 : Bool;
               x03 : Bool;
               x04 : Bool;
               x05 : Bool;
               x06 : Bool;
               x07 : Bool;
            END_STRUCT;
         END_STRUCT;
      END_STRUCT;
      read2 : Struct
         fault_contents_1 : Struct
            x08_inverter_overheat : Bool;
            x09_inverter_overheat_warning : Bool;
            x10_motor_overload : Bool;
            x11_inverter_overload : Bool;
            x12_overtorque_1 : Bool;
            x13_overtorque_2 : Bool;
            x14_braking_resistor_fault : Bool;
            x15_braking_resistor_overheat : Bool;
            x00_fuse : Bool;
            x01_main_circuit_undervoltage : Bool;
            x02_control_circuit_undervoltage : Bool;
            x03_mc_error : Bool;
            x04 : Bool;
            x05_ground_fault : Bool;
            x06_over_current : Bool;
            x07_overvoltage : Bool;
            "a" : Struct
               x08 : Bool;
               x09 : Bool;
               x10 : Bool;
               x11 : Bool;
               x12 : Bool;
               x13 : Bool;
               x14 : Bool;
               x15 : Bool;
               x00 : Bool;
               x01 : Bool;
               x02 : Bool;
               x03 : Bool;
               x04 : Bool;
               x05 : Bool;
               x06 : Bool;
               x07 : Bool;
            END_STRUCT;
         END_STRUCT;
      END_STRUCT;
      read3_data : Struct
         "Output Frequency" : Word;   // 0.01Hz
         "Output Current" : Word;   // 0.1A
         "Output Voltage" : Word;   // 0.1Vac
         "DC Bus Voltage" : Word;   // Vdc
         "Output Power" : Word;   // 0.1kW
      END_STRUCT;
      _ : Bool;
      write1 : Struct
         cmd : Struct
            x08 : Bool;
            x09 : Bool;
            x10 : Bool;
            x11 : Bool;
            x12 : Bool;
            x13 : Bool;
            x14 : Bool;
            x15 : Bool;
            x00_run : Bool := TRUE;
            x01_reverse : Bool;
            x02_external_fault : Bool;
            x03_fault_reset : Bool;
            x04_ComNet : Bool := TRUE;
            x05_ComCtrl : Bool := TRUE;
            x06 : Bool;
            x07 : Bool;
         END_STRUCT;
         freq_ref : Int;
      END_STRUCT;
      write2_max_frequency : UInt := 50;   // 0.1 Hz
      write3 : Struct
         ref_source : Int := 2;   // 0=Operator, 1=Terminals, 2=Serial Com, 3=Option PCB
         run_source : Int := 2;   // 0=Operator, 1=Terminals, 2=Serial Com, 3=Option PCB
         stopp_method : Int := 0;   // 0=Ramp to Stop, 1=Coast to Stop, 2=DCInj to Stop, 3=Coast w/Timer (C1-09)
      END_STRUCT;
   END_VAR
BEGIN
   // Yaskawa - E7 Drive
   // Models: CIMR-E7U* 
   // Web: https://www.ccontrols.com/support/dp/TME711.pdf

   "mb_station_block_header"(sb := #sb,
                             mb_query := #mb_query);
   #mb_query.mb_addr := #mb_addr;

   #mb_query.mode := #mb_query.c.read.holding_reg;
   #mb_query(data_addr := 16#10,
             data_ptr := #read1);
   #mb_query(data_addr := 16#14,
             data_ptr := #read2);
   #mb_query(data_addr := 16#41,
             data_ptr := #read3_data);

   #mb_query.mode := #mb_query.c.write.holding_reg;
   #mb_query(data_addr := 16#303,
             data_ptr := #write2_max_frequency);
   #mb_query(data_addr := 16#180,
             data_ptr := #write3);
   #mb_query(data_addr := 16#1,
             data_ptr := #write1);

   "mb_station_block_footer"(sb := #sb,
                             mb_query := #mb_query);
END_FUNCTION_BLOCK

FUNCTION_BLOCK "Yokogawa_multivariable_transmitter"   // FB77, SCL
{ S7_Optimized_Access := 'TRUE' }
VERSION : 0.1
   VAR_INPUT
      mb_addr : UInt;
   END_VAR
   VAR_IN_OUT
      mb_query : "mb_query";
   END_VAR
   VAR
      sb : "mb_station_block_udt";
      data : Struct
         pres : Real;
         sp : Real;
         et : Real;
      END_STRUCT;
   END_VAR
BEGIN
   // Yokogawa - EJX910A and EJX930A - Multivariable Transmitter
   // web: https://web-material3.yokogawa.com/IM01C25R05-01EN_001.pdf?_ga=
   //      2.43421607.346053457.1505559574-1218156352.1505559574

   "mb_station_block_header"(sb := #sb, mb_query := #mb_query);
   #mb_query.mb_addr := #mb_addr;

   #mb_query(mode := #mb_query.c.read.input_reg,
             data_addr := 401,
             data_ptr := #data);

   "mb_station_block_footer"(sb := #sb, mb_query := #mb_query);
END_FUNCTION_BLOCK

FUNCTION_BLOCK "Accuenergy_Accuvim_L_Series_Power_meter"   // FB81, SCL
{ S7_Optimized_Access := 'TRUE' }
VERSION : 0.1
   VAR_INPUT
      mb_addr : USInt;
   END_VAR
   VAR_IN_OUT
      mb_query : "mb_query";
   END_VAR
   VAR
      sb : "mb_station_block_udt";
      read1 : Struct
         Frequency : Real;
         "Phase voltage" : Array[1..3] of Real;
         "Line voltage" : Array[1..3] of Real;
         Phase_current : Array[1..3] of Real;
         Neutral_current : Real;
         "Phase power" : Array[1..3] of Real;
         "System power Psum" : Real;
         "Phase reactive power" : Array[1..3] of Real;
         "System reactive power" : Real;
         "System apparent Ssum" : Real;
         Phase_power_factor : Array[1..3] of Real;
         "System power PFsum" : Real;
         "Voltage unbalance factor" : Real;
         "Current unbalance factor" : Real;
         _ : DWord;
         "Phase apparent power S" : Array[1..3] of Real;
         __ : DWord;
         "Apparent power demand" : Real;
         "Power demand P_Dmd" : Real;
         "Reactive power demand" : Real;
         "Phase current demand" : Array[1..3] of Real;
      END_STRUCT;
      read2_run_time : Struct
         Meter : UDInt;
         Load : UDInt;
      END_STRUCT;
      read3 : Struct
         Import_energy_Ep_imp : UDInt;
         Export_energy_Ep_exp : UDInt;
         Import_reactive_energy_Eq_imp : UDInt;
         Export_reactive_energy_Eq_exp : UDInt;
         Apparent_energy_Es : UDInt;
         Phase_energy : Array[1..3] of Struct
            "import Ep_imp" : UDInt;
            "export Ep_exp" : UDInt;
         END_STRUCT;
      END_STRUCT;
   END_VAR
BEGIN
   // Accuenergy - Accuvim-L Series Power meter
   // 
   // - https://www.accuenergy.com/files/acuvim-l/
   //   Acuvim-L-Panel-Submeter-Power-Energy-Meter-User-%20Manual(1030E2201).pdf

   "mb_station_block_header"(sb := #sb,
                             mb_query := #mb_query);
   #mb_query.mb_addr := #mb_addr;

   #mb_query.mode := #mb_query.c.read.holding_reg;
   #mb_query(data_addr := 16#600,
             data_ptr := #read1);
   #mb_query(data_addr := 16#180,
             data_ptr := #read2_run_time);
   #mb_query(data_addr := 16#156,
             data_ptr := #read3);

   "mb_station_block_footer"(sb := #sb,
                             mb_query := #mb_query);
END_FUNCTION_BLOCK

FUNCTION_BLOCK "DAE_Instrument_PM210"   // FB82, SCL
{ S7_Optimized_Access := 'TRUE' }
VERSION : 0.1
   VAR_INPUT
      mb_addr : USInt;
   END_VAR
   VAR_IN_OUT
      mb_query : "mb_query";
   END_VAR
   VAR
      sb : "mb_station_block_udt";
   END_VAR
   VAR RETAIN
      conf : Struct
         write : Bool;
         PT_ratio : Real;
         CT_ratio : Real;
      END_STRUCT;
   END_VAR
   VAR
      data1 : Struct
         voltage_Lx_N : Array[1..3] of Real;
         voltage_L_L : Array[1..3] of Real;
         current : Array[1..3] of Real;
         total_active_power : Real;
         total_reactive_power : Real;
         total_apparent_power : Real;
         frequency : Real;
         power_factor : Real;
         total_active_energy : Real;
         total_reactive_energy : Real;
         "15_minute_block_demand" : Real;
         "1_minute_block_demand" : Real;
         generator_total_active_energy : Real;
         generator_total_reactive_energy : Real;
      END_STRUCT;
      data2 : Struct
         energy_active : Struct   // VA
            phase : Array[1..3] of Real;
            total : Real;
         END_STRUCT;
         energy_reactive : Struct
            phase : Array[1..3] of Real;
            total : Real;
         END_STRUCT;
         power_active : Struct
            phase : Array[1..3] of Real;
            total : Real;
         END_STRUCT;
         power_reactive : Struct
            phase : Array[1..3] of Real;
            total : Real;
         END_STRUCT;
         power_apparent : Struct
            phase : Array[1..3] of Real;
            total : Real;
         END_STRUCT;
         power_factor : Struct
            phase : Array[1..3] of Real;
            total : Real;
         END_STRUCT;
      END_STRUCT;
      read3_temperature : Int;
      read4_io : Struct
         digital_output : Word;
         digital_input : Word;
      END_STRUCT;
      data5_generator_energy : Struct
         active : Struct
            phase : Array[1..3] of Real;
            total : Real;
         END_STRUCT;
         reactive : Struct
            phase : Array[1..3] of Real;
            total : Real;
         END_STRUCT;
      END_STRUCT;
   END_VAR
   VAR_TEMP
      read1 : Struct
         voltage_Lx_N : Array[1..3] of UDInt;   // volt
         voltage_L_L : Array[1..3] of UDInt;   // volt 1:L1-L2, 2:L2-L3, 3:L3-L1
         current : Array[1..3] of UDInt;   // mA
         total_active_power : UDInt;
         total_reactive_power : UDInt;
         total_apparent_power : UDInt;
         frequency : UDInt;
         power_factor : DInt;
         total_active_energy : UDInt;
         total_reactive_energy : UDInt;
         "15_minute_block_demand" : UDInt;
         "1_minute_block_demand" : UDInt;
         generator_total_active_energy : UDInt;
         generator_total_reactive_energy : UDInt;
      END_STRUCT;
      read2 : Struct
         energy_active : Struct   // VA
            phase : Array[1..3] of UDInt;
            total : UDInt;
         END_STRUCT;
         energy_reactive : Struct
            phase : Array[1..3] of UDInt;
            total : UDInt;
         END_STRUCT;
         power_active : Struct
            phase : Array[1..3] of UDInt;
            total : UDInt;
         END_STRUCT;
         power_reactive : Struct
            phase : Array[1..3] of UDInt;
            total : UDInt;
         END_STRUCT;
         power_apparent : Struct
            phase : Array[1..3] of UDInt;
            total : UDInt;
         END_STRUCT;
         power_factor : Struct
            phase : Array[1..3] of Int;
            total : Int;
         END_STRUCT;
      END_STRUCT;
      read5_generator_energy : Struct
         active : Struct
            phase : Array[1..3] of UDInt;
            total : UDInt;
         END_STRUCT;
         reactive : Struct
            phase : Array[1..3] of UDInt;
            total : UDInt;
         END_STRUCT;
      END_STRUCT;
      write1 : Struct
         PT_ratio : UInt;
         CT_ratio : UInt;
      END_STRUCT;
      c : Int;
   END_VAR
BEGIN
   // DAE Instrument Corp. - PM210 
   // Multi-Function Panel Meter
   //
   // Default: 9600-8-N-1
   // 
   // http://www.daeinstrument.com/downloads/PM210%20Modbus%20Reference-2.6.1e.pdf

   "mb_station_block_header"(sb := #sb, mb_query := #mb_query);
   #mb_query.mb_addr := #mb_addr;
   #mb_query.mode := #mb_query.c.read.holding_reg;

   #mb_query(data_addr := 20, data_ptr := #read1);
   IF #mb_query.Done THEN
       FOR #c := 1 TO 3 DO
           #data1.voltage_Lx_N[#c] := UDINT_TO_REAL(ROR(IN := #read1.voltage_Lx_N[#c], N := 16)) * 0.1;
           #data1.voltage_L_L[#c] := UDINT_TO_REAL(ROR(IN := #read1.voltage_L_L[#c], N := 16)) * 0.1;
           #data1.current[#c] := UDINT_TO_REAL(ROR(IN := #read1.current[#c], N := 16)) * 0.001;
       END_FOR;
       #data1.total_active_power := UDINT_TO_REAL(ROR(IN := #read1.total_active_power, N := 16));
       #data1.total_reactive_power := UDINT_TO_REAL(ROR(IN := #read1.total_reactive_power, N := 16));
       #data1.total_apparent_power := UDINT_TO_REAL(ROR(IN := #read1.total_apparent_power, N := 16));
       #data1.frequency := UDINT_TO_REAL(ROR(IN := #read1.frequency, N := 16)) * 0.1;
       #data1.power_factor := DINT_TO_REAL(ROR(IN := #read1.power_factor, N := 16)) * 0.001;
       #data1.total_active_energy := UDINT_TO_REAL(ROR(IN := #read1.total_active_energy, N := 16)) * 0.01;
       #data1.total_reactive_energy := UDINT_TO_REAL(ROR(IN := #read1.total_reactive_energy, N := 16)) * 0.01;
       #data1."15_minute_block_demand" := UDINT_TO_REAL(ROR(IN := #read1."15_minute_block_demand", N := 16)) * 0.1;
       #data1."1_minute_block_demand" := UDINT_TO_REAL(ROR(IN := #read1."1_minute_block_demand", N := 16)) * 0.1;
       #data1.generator_total_active_energy := UDINT_TO_REAL(ROR(IN := #read1.generator_total_active_energy, N := 16)) * 0.01;
       #data1.generator_total_reactive_energy := UDINT_TO_REAL(#read1.generator_total_reactive_energy) * 0.01;
   END_IF;

   #mb_query(data_addr := 80, data_ptr := #read2);
   IF #mb_query.Done THEN
       FOR #c := 1 TO 3 DO
           #data2.energy_active.phase[#c] := UDINT_TO_REAL(ROR(IN := #read2.energy_active.phase[#c], N := 16)) * 0.01;
           #data2.energy_reactive.phase[#c] := UDINT_TO_REAL(ROR(IN := #read2.energy_reactive.phase[#c], N := 16)) * 0.01;
           #data2.power_active.phase[#c] := UDINT_TO_REAL(ROR(IN := #read2.power_active.phase[#c], N := 16));
           #data2.power_reactive.phase[#c] := UDINT_TO_REAL(ROR(IN := #read2.power_reactive.phase[#c], N := 16));
           #data2.power_apparent.phase[#c] := UDINT_TO_REAL(ROR(IN := #read2.power_apparent.phase[#c], N := 16));
           #data2.power_factor.phase[#c] := INT_TO_REAL(#read2.power_factor.phase[#c]) * 0.001;
       END_FOR;
       #data2.energy_active.total := UDINT_TO_REAL(ROR(IN := #read2.energy_active.total, N := 16)) * 0.01;
       #data2.energy_reactive.total := UDINT_TO_REAL(ROR(IN := #read2.energy_reactive.total, N := 16)) * 0.01;
       #data2.power_active.total := UDINT_TO_REAL(ROR(IN := #read2.power_active.total, N := 16));
       #data2.power_reactive.total := UDINT_TO_REAL(ROR(IN := #read2.power_reactive.total, N := 16));
       #data2.power_apparent.total := UDINT_TO_REAL(ROR(IN := #read2.power_apparent.total, N := 16));
       #data2.power_factor.total := INT_TO_REAL(#read2.power_factor.total) * 0.001;
   END_IF;

   #mb_query(data_addr := 139, data_ptr := #read3_temperature);
   #mb_query(data_addr := 142, data_ptr := #read4_io);
   #mb_query(data_addr := 144, data_ptr := #read5_generator_energy);
   IF #mb_query.Done THEN
       FOR #c := 1 TO 3 DO
           #data5_generator_energy.active.phase[#c] := UDINT_TO_REAL(ROR(IN := #read5_generator_energy.active.phase[#c], N := 16)) * 0.01;
           #data5_generator_energy.reactive.phase[#c] := UDINT_TO_REAL(ROR(IN := #read5_generator_energy.reactive.phase[#c], N := 16)) * 0.01;
       END_FOR;
       #data5_generator_energy.active.total := UDINT_TO_REAL(ROR(IN := #read5_generator_energy.active.total, N := 16)) * 0.01;
       #data5_generator_energy.reactive.total := UDINT_TO_REAL(ROR(IN := #read5_generator_energy.reactive.total, N := 16)) * 0.01;
   END_IF;

   IF #conf.write THEN
       #write1.PT_ratio := REAL_TO_UINT(#conf.PT_ratio * 100);
       #write1.CT_ratio := REAL_TO_UINT(#conf.CT_ratio);
       #mb_query(mode := #mb_query.c.write.holding_reg,
                 data_addr := 133,
                 data_ptr := #write1);
       #conf.write := #conf.write AND NOT #mb_query.Done;
   END_IF;

   "mb_station_block_footer"(sb := #sb, mb_query := #mb_query);
END_FUNCTION_BLOCK

FUNCTION_BLOCK "Integron_OXY-DIOS-DSP"   // FB84, SCL
{ S7_Optimized_Access := 'TRUE' }
VERSION : 0.1
   VAR_INPUT
      mb_addr : USInt;
   END_VAR
   VAR_IN_OUT
      mb_query : "mb_query";
   END_VAR
   VAR
      sb : "mb_station_block_udt";
      read1 : Struct
         Sensor_status : Struct
            x08 : Bool;
            x09 : Bool;
            x10 : Bool;
            x11 : Bool;
            x12 : Bool;
            x13 : Bool;
            x14 : Bool;
            x15 : Bool;
            x00_Correct_indication : Bool;
            x01_Range_exceeded_error : Bool;
            x02_Measuring_window_status : Bool;   // (Must be replaced)
            x03_Cleaning : Bool;
            x04_Maintaining_values_after_cleaning : Bool;   // ("holding time") F= Real current value, T=Saved value
            x05_Output_short_circuit_OXYGEN_CONTROL : Bool;
            x06_Output_short_circuit_AIRBLAST_CLEANING : Bool;
            x07 : Bool;
         END_STRUCT;
         cO2_concentration : Real;   // [mg/L]
         sO2_saturation : Real;   // [%]
         Head_temperature : Real;   // [degree C]
         pO2_O2_partial_pressure : Real;   // [bar]
         Tau_fluorescence_decay_time : Real;   // [us]
         Atmospheric_pressure : Real;   // [bar] (hydrostatic)
         Relative_humidity_inside_the_sensor : Real;   // [%]
         Humidity_sensor_temperature : Real;   // [degree C]
         Salinity : Real;   // [ppt]
         Mainboard_temperature : Real;   // [degree C]
         Sensor_serial_number : Array[1..4] of Word;
         Date_and_time : UDInt;   // [s]
         Window_serial_number : UInt;
         Expected_date_of_exchange_measuring_window : UDInt;   // [s]
         Date_of_last_calibration : UDInt;   // [s]
         RTC_battery_level : UInt;   // [%]
         Supply_power_24V : Real;
      END_STRUCT;
   END_VAR
BEGIN
   // Integron Poland EU - OXY-DIOS-DSP
   // Optical dissolved oxygen sensor
   // 
   // https://www.tme.eu/en/Document/9d0bf7a4d6041739cc6d58df1cc838cb/OXY-DIOS-DSP-Manual-EN-v.1.33.pdf
   // http://www.sensor.integron.pl

   "mb_station_block_header"(sb := #sb, mb_query := #mb_query);
   #mb_query.mb_addr := #mb_addr;

   #mb_query.mode := #mb_query.c.mode.read;
   #mb_query(data_addr := 41000, data_ptr := #read1);

   "mb_station_block_footer"(sb := #sb, mb_query := #mb_query);
END_FUNCTION_BLOCK

FUNCTION_BLOCK "masibus_85XX"   // FB86, SCL
{ S7_Optimized_Access := 'TRUE' }
VERSION : 0.1
   VAR_INPUT
      mb_addr : USInt;
   END_VAR
   VAR_IN_OUT
      mb_query : "mb_query";
   END_VAR
   VAR
      sb : "mb_station_block_udt";
      read1 : Struct
         channel : Array[1..24] of Int;
         Ambient_PV : Int;
         digital_output_status : DWord;
         alarm : Array[1..2] of DWord;
         control_status : DWord;
         alarm_blink_status : Array[1..2] of DWord;
         alarm_LED_status : Array[1..2] of DWord;
      END_STRUCT;
      write1_labels : Array[1..24] of String[6];
      write2_input_type : Array[1..24] of USInt;
   END_VAR
BEGIN
   // Masibus - 85XX+
   // SCANNER / DAQ
   // REF NO: m83B/om/101
   // http://www.masibus.com/Pmanual/Data_Acquisition/
   // Enhanced_Multi-Channel_Scanners/85XX+_User_Manual

   "mb_station_block_header"(sb := #sb,
                             mb_query := #mb_query);
   #mb_query.mb_addr := #mb_addr; // Device address.

   #mb_query.mode := #mb_query.c.mode.read;
   #mb_query(data_addr := 30001,
             data_ptr := #read1);

   #mb_query.mode := #mb_query.c.mode.write;
   #mb_query(data_addr := 42204,
             data_ptr := #write1_labels);
   #mb_query(data_addr := 40097,
             data_ptr := #write2_input_type);

   "mb_station_block_footer"(sb := #sb,
                             mb_query := #mb_query);

   (*

   #  : Type
   ------------
   00 : None
   01 : E-tc
   02 : J-tc
   03 : K-tc
   04 : T-tc
   05 : B-tc
   06 : R-tc 
   07 : S-tc
   08 : n-tc
   09 : RDT
   10 : Cu53
   11 : Ni120
   12 : -10.20mV
   13 : 0-100mV
   14 : 4-20mA
   15 : 0-20mA
   16 : 0-5V
   17 : 1-5V
   18 : 0-10V
   19 : Dig.inp

   *)
END_FUNCTION_BLOCK

// folder: Library/Modbus/Station blocks/Abb

FUNCTION_BLOCK "abb_aquaMaster_3"   // FB4, SCL
{ S7_Optimized_Access := 'TRUE' }
VERSION : 0.1
   VAR_INPUT
      mb_addr : USInt;
   END_VAR
   VAR_IN_OUT
      mb_query : "mb_query";
   END_VAR
   VAR
      sb : "mb_station_block_udt";
      flow : Real;
      pressure : Real;
      totaliser : Struct
         fwd : DInt;
         rev : DInt;
         net : DInt;
      END_STRUCT;
   END_VAR
BEGIN
   // - ABB - AquaMaster 3 - Electromagnetic flowmeter
   // - COI/FET2XX/MOD/TBLÃ¢â‚¬â€œEN
   // - https://library.e.abb.com/public/
   //   91eead459bb0d349c12577fc0033d2b5/COI_FET2XX_MOD_TBL-EN.pdf

   "mb_station_block_header"(sb := #sb, mb_query := #mb_query);
   #mb_query.mb_addr := #mb_addr; // Device address.

   // Two queries, reading input registers. 
   #mb_query.mode := #mb_query.c.read.input_reg;
   #mb_query(data_addr := 5017, data_ptr := #flow);
   #mb_query(data_addr := 5025, data_ptr := #pressure);

   // One query, reading one section of holding registers.
   #mb_query.mode := #mb_query.c.read.holding_reg;
   #mb_query(data_addr := 12003, data_ptr := #totaliser);

   // - Each query reading one section of holding registers.
   // - Data length is automatically calculated for holding 
   //   and input regisers.

   "mb_station_block_footer"(sb := #sb, mb_query := #mb_query);
END_FUNCTION_BLOCK

FUNCTION_BLOCK "Abb_266"   // FB12, SCL
{ S7_Optimized_Access := 'TRUE' }
VERSION : 0.1
   VAR_INPUT
      mb_addr : UInt;
   END_VAR
   VAR_IN_OUT
      mb_query : "mb_query";
   END_VAR
   VAR
      sb : "mb_station_block_udt";
      data : Struct
         "Differential Pressure" : Real;
         "Static Pressure" : Real;
         "Process Temperature" : Real;
         "Mass flow rate value" : Real;
         "Volume Flow rate value" : Real;
      END_STRUCT;
      settings : Struct
         Differential_Pressure_Units_Code : UInt := 12;
         Static_Pressure_Units_select_Code : UInt := 12;
         Temperature_Units_select_Code : UInt := 32;
      END_STRUCT;
   END_VAR
BEGIN
   // ABB - 266 MODBUS, multivariable transmitter.
   // Differential and Static Pressure, Temperature
   // 
   // https://library.e.abb.com/public/9b5a1233ec79400387d5b4887002fb00/2105216MNAA.pdf

   "mb_station_block_header"(sb := #sb, mb_query := #mb_query);
   #mb_query.mb_addr := #mb_addr;

   #mb_query(mode := #mb_query.c.read.holding_reg,
             data_addr := 401,
             data_ptr := #data);

   #mb_query(mode := #mb_query.c.write.holding_reg,
             data_addr := 481,
             data_ptr := #settings);

   "mb_station_block_footer"(sb := #sb, mb_query := #mb_query);

   (*
   Differential_Pressure_Units_Code
   1 = inches of water
   8 = Millibar (ROM default)
   11 = Pascal
   12 = Kilopascal 

   Static Pressure Units select Code
   6 = PSIA
   7 = Bar (ROM default)
   12 = Kilopascal
   117 = Megapascal 

   Temperature Units select Code
   32 = Degree Celsius (ROM default)
   33 = Degree Fahrenheit
   34 = Degree Rankine
   35 = Degree Kelvin

   *)
END_FUNCTION_BLOCK

FUNCTION_BLOCK "Abb_M2M_DMTME"   // FB15, SCL
{ S7_Optimized_Access := 'TRUE' }
VERSION : 0.1
   VAR_INPUT
      mb_addr : UInt;
   END_VAR
   VAR_IN_OUT
      mb_query : "mb_query";
   END_VAR
   VAR
      sb : "mb_station_block_udt";
      read1 : Struct
         "3-PHASE SYSTEM VOLTAGE" : UDInt;   // volt
         voltage_Lx_N : Array[1..3] of UDInt;   // volt
         voltage_L_L : Array[1..3] of UDInt;   // volt 1:L1-L2, 2:L2-L3, 3:L3-L1
         "3-PHASE SYSTEM CURRENT" : UDInt;
         current : Array[1..3] of UDInt;   // mA
         "3-PHASE SYS. POWER FACTOR" : DInt;   // x1000
         Power_factor : Array[1..3] of DInt;   // x1000
         "3-PHASE SYSTEM COS Ï•I" : DInt;   // x1000
         phase_cos : Array[1..3] of DInt;   // x1000
      END_STRUCT;
      read2 : Struct
         "3-PHASE S. APPARENT POWER" : UDInt;   // VA
         apparent_power : Array[1..3] of UDInt;   // VA
         "3-PHASE SYS. ACTIVE POWER" : DInt;   // Watt
         active_power : Array[1..3] of DInt;   // Watt
         "3-PHASE S. REACTIVE POWER" : UDInt;
         reactive_power : Array[1..3] of UDInt;
         "3-PHASE SYS. ACTIVE ENERGY" : UDInt;   // Wh * 100
         "3-PHASE S. REACTIVE ENERGY" : UDInt;   // VArh * 100
         frequency : UDInt;   // mHz
         "MAX LINE CURRENT" : Array[1..3] of UDInt;
      END_STRUCT;
   END_VAR
BEGIN
   // ABB - M2M/DMTME - 2CSG445011D0201 
   //
   // https://library.e.abb.com/public/3921770555944801ad6d9e002d23ca23/2CSG445011D0201.pdf

   "mb_station_block_header"(sb := #sb, mb_query := #mb_query);
   #mb_query.mb_addr := #mb_addr;

   #mb_query.mode := #mb_query.c.read.holding_reg;
   #mb_query(data_addr := 16#1000, data_ptr := #read1);
   #mb_query(data_addr := 16#1026, data_ptr := #read2);

   "mb_station_block_footer"(sb := #sb, mb_query := #mb_query);
END_FUNCTION_BLOCK

FUNCTION_BLOCK "Abb_ach_400_ac_drives"   // FB80, SCL
{ S7_Optimized_Access := 'TRUE' }
VERSION : 0.1
   VAR_INPUT
      mb_addr : UInt;
   END_VAR
   VAR_IN_OUT
      mb_query : "mb_query";
   END_VAR
   VAR
      sb : "mb_station_block_udt";
      read1 : Struct
         sw : Struct   // page 111, tabel 23
            x08_actual_eq_ref : Bool;   // (= is within tolerance limits)
            x09_drive_control_remote : Bool;
            x10_supervision_limit : Bool;   // The value of first supervised parameter equals to or is greater than supervision limit. Refer toGroup 32 Supervision.
            x11_ext2_selected : Bool;   // 0 = ext1 selected
            x12_run : Bool;   // Enable signal received
            x13 : Bool;
            x14 : Bool;
            x15 : Bool;
            x00_rdy_to_sw_on : Bool;
            x01_rdy_to_operate : Bool;
            x02_opr_enabled : Bool;
            x03_falut : Bool;
            x04_OFF2_inactive : Bool;
            x05_OFF3_inactive : Bool;
            x06_switch_on_innhibited : Bool;
            x07_alarm : Bool;   // See the Diagnostics section for a list of relevant alarms
         END_STRUCT;
      END_STRUCT;
      read2 : Struct
         speed : Int;   // rpm
         output_freq : Int;   // 0.1 Hz
         current : Int;   // 0.1 A
         torque : Int;   // 0.1 %
         power : Int;   // 0.1 kW
         dc_bus_voltage : Int;   // 0.1 V
         output_voltage : Int;   // 0.1 V
         ACH400_temp : Int;   // 0.1 Â°C | Displays the temperature of the ACH 400 heatsink in degrees Centigrade
         ext_ref_1 : Int;   // 0.1 Hz
         ext_ref_2 : Int;   // 0.1 %
         ctrl_location : Int;   // 0 - 2
         run_time : UInt;   // h
         kWh_cnt : UInt;   // kWh
         appl_blk_output : UInt;
         digital_input : Struct
            x08 : Bool;
            x09 : Bool;
            x10 : Bool;
            x11 : Bool;
            x12 : Bool;
            x13 : Bool;
            x14 : Bool;
            x15 : Bool;
            x00_in_1 : Bool;
            x01_in_2 : Bool;
            x02_in_3 : Bool;
            x03_in_4 : Bool;
            x04 : Bool;
            x05 : Bool;
            x06 : Bool;
            x07 : Bool;
         END_STRUCT;
         analog_in_1 : UInt;   // 0.1 %
         analog_in_2 : UInt;   // 0.1 %
      END_STRUCT;
      read3 : Struct
         fault_word_1 : Struct
            x08_Motor_overtemperature : Bool;
            x09_Panel_loss : Bool;
            x10_Parameters_inconsistent : Bool;
            x11_DC_bus_ripple_too_large : Bool;
            x12_Motor_stall : Bool;
            x13_Serial_communication_loss : Bool;
            x14_External_fault : Bool;
            x15_Output_ground_fault : Bool;
            x00_Overcurrent : Bool;
            x01_DC_overvoltage : Bool;
            x02_ACH_400_overtemperature : Bool;
            x03_Fault_current : Bool;
            x04_Output_overload : Bool;
            x05_DC_undervoltage : Bool;
            x06_Analog_input_1_fault : Bool;
            x07_Analog_input_2_fault : Bool;
         END_STRUCT;
         fault_word_2 : Struct
            x08_hw_err : Bool;
            x09_hw_err : Bool;
            x10_hw_err : Bool;
            x11_hw_err : Bool;
            x12_hw_err : Bool;
            x13_hw_err : Bool;
            x14_hw_err : Bool;
            x15_hw_err : Bool;
            x00_Underload : Bool;
            x01 : Bool;
            x02_DDCS_link : Bool;
            x03 : Bool;
            x04 : Bool;
            x05 : Bool;
            x06 : Bool;
            x07 : Bool;
         END_STRUCT;
      END_STRUCT;
      _ : Bool;
      write1 : Struct
         cw : Struct   // page 109, tabel 21
            x08 : Bool;
            x09 : Bool;
            x10 : Bool;
            x11_sel_ext_2 : Bool;   // Select external control location 1
            x12 : Bool;
            x13 : Bool;
            x14 : Bool;
            x15 : Bool;
            x00_start : Bool := TRUE;
            x01_no_cost_stop : Bool := TRUE;   // Emergency OFF, coast to stop.Enter OFF2 ACTIVE; proceed to SWITCH-ON INHIBITED
            x02_no_ramp_stop : Bool := TRUE;   // Emergency stop. Drive ramps to stop according to parameter 2205 DECELER TIME 2. Enter
            x03_operation_enable : Bool := TRUE;
            x04 : Bool;
            x05_no_ramp_generator : Bool := TRUE;
            x06_no_force_ramp_generator_input2zero : Bool;   // Force Ramp Function Generator input to zero
            x07_fault_reset : Bool;   // (enter SWITCH-ON INHIBITED)
         END_STRUCT;
         ref_1 : Int;
         ref_2 : Int;
      END_STRUCT;
      write2 : Struct
         keypad_ref_sel : UInt;
         ext1_ext2_sel : UInt;
         ext1_sel : UInt;
         ext1_sel_min : UInt;   // 0 - 250 Hz
         ext1_sel_max : UInt := 50;   // 0 - 250 Hz
      END_STRUCT;
      write3 : Struct   // Communication fault function
         comm_fault_func : UInt := 1;   // 1=FAULT(cost), 2=CONST SP 7, 3=LAST SPEED
      END_STRUCT;
   END_VAR
BEGIN
   // Abb - ACH 400 - AC Drives 
   // 
   // Web: https://www.ccontrols.com/support/dp/ACH402_US_04_Web.pdf

   "mb_station_block_header"(sb := #sb, mb_query := #mb_query);
   #mb_query.mb_addr := #mb_addr;

   #mb_query.mode := #mb_query.c.read.holding_reg;
   #mb_query(data_addr := 3, data_ptr := #read1);   // 40004
   #mb_query(data_addr := 102, data_ptr := #read2); // 103
   #mb_query(data_addr := 304, data_ptr := #read3); // 305 - 1 

   #mb_query.mode := #mb_query.c.write.holding_reg;
   #mb_query(data_addr := 0, data_ptr := #write1); // 40001
   // #mb_query(data_addr := 1100, data_ptr := #write2); // 1101 - 1
   #mb_query(data_addr := 5003, data_ptr := #write3); // 5004 - 1

   "mb_station_block_footer"(sb := #sb, mb_query := #mb_query);
END_FUNCTION_BLOCK

// folder: Library/Modbus/Station blocks/Floridan

FUNCTION_BLOCK "Floridan_Uniflo_1200"   // FB83, SCL
{ S7_Optimized_Access := 'TRUE' }
VERSION : 0.1
   VAR_INPUT
      mb_addr : USInt;
      delay : Time := T#10S;
   END_VAR
   VAR_OUTPUT
      energi : LReal;   // [MJ]
      vol_measured : LReal;   // [m3]
      vol_conv : LReal;   // [Nm3]
      pressure : LReal;   // [bar A]
      temperature : LReal;
   END_VAR
   VAR_IN_OUT
      mb_query : "mb_query";
   END_VAR
   VAR
      sb : "mb_station_block_udt";
      battery_remaining : UInt;
      mb_delay : "mb_delay";
      serial_number : String[6];
   END_VAR
   VAR_TEMP
      dommy : Bool;
      c : Int;
      "dword" : DWord;
   END_VAR
BEGIN
   // Flonidan - Uniflo 1200 GVEC
   // Product number: 061864X-YYY
   //
   // - https://www.gavilar.nl/files/communicationboard230210_1521630740_b6a3b533.pdf
   // - M/06180XX/24

   "mb_station_block_header"(sb := #sb, mb_query := #mb_query);
   #mb_query.mb_addr := #mb_addr; // Device address.

   // Reduce power consumption, by halting execution. Nice if the device is running 
   // on battery. mb_delay is located inside the mb_extended_features.scl file.
   #mb_delay(delay := #delay, mb_query := #mb_query);

   #mb_query.mb_addr.%X5 := 0; // - Last bits of mb_addr is used for expanding 
   #mb_query.mb_addr.%X6 := 0; //   register addr, this means that only addr 1
   #mb_query.mb_addr.%X7 := 0; //   to 31 on the bus may be used.

   #mb_query.mode := #mb_query.c.read.holding_reg;

   #mb_query(data_addr := 123, data_ptr := #battery_remaining);
   #mb_query(data_addr := 2833, data_ptr := #serial_number); // Serial number 

   #mb_query.conf.buffer_handler := false;

   #mb_query(data_addr := 56, data_len := 44, data_ptr := #dommy);
   IF #mb_query.Done THEN
       #vol_conv := "intreal"(mb_query := #mb_query, addr := 16#70 / 2);
       #"dword".%B3 := #mb_query.z.buffer[16]; // 16#80/2=64, (64-56)*2=16
       #"dword".%B2 := #mb_query.z.buffer[17];
       #"dword".%B1 := #mb_query.z.buffer[18];
       #"dword".%B0 := #mb_query.z.buffer[19];
       #pressure := DWORD_TO_REAL(#"dword");
       #"dword".%B3 := #mb_query.z.buffer[20]; // 16#84/2=66, (66-56)*2=20
       #"dword".%B2 := #mb_query.z.buffer[21];
       #"dword".%B1 := #mb_query.z.buffer[22];
       #"dword".%B0 := #mb_query.z.buffer[23];
       #temperature := DWORD_TO_REAL(#"dword");
       #energi := "intreal"(mb_query := #mb_query, addr := 16#90 / 2);
       #vol_measured := "intreal"(mb_query := #mb_query, addr := 16#98 / 2);
   END_IF;

   #mb_query.data_len := #mb_query.c.auto_len;
   #mb_query.conf.buffer_handler := true;
   "mb_station_block_footer"(sb := #sb, mb_query := #mb_query);
END_FUNCTION_BLOCK

FUNCTION "intreal" : LReal   // FC16, SCL
{ S7_Optimized_Access := 'TRUE' }
VERSION : 0.1
   VAR_INPUT
      mb_query : "mb_query";
      addr : UInt;
   END_VAR
   VAR_TEMP
      dw : UDInt;
      r : DWord;
      bo : UDInt;
   END_VAR
BEGIN
   // Uniflo 1200 has a special datatype named
   // int-real, this block decode that data type.

   // buffer offset
   #bo := (#addr - #mb_query.data_addr) * 2;

   // The integer part of the value, little endian.
   #dw.%B3 := #mb_query.z.buffer[#bo + 0];
   #dw.%B2 := #mb_query.z.buffer[#bo + 1];
   #dw.%B1 := #mb_query.z.buffer[#bo + 2];
   #dw.%B0 := #mb_query.z.buffer[#bo + 3];
   #intreal := UDINT_TO_LREAL(#dw);

   // The decimal part of the value, little endian.
   // Stored as a real (IEEE754).
   #r.%B3 := #mb_query.z.buffer[#bo + 4];
   #r.%B2 := #mb_query.z.buffer[#bo + 5];
   #r.%B1 := #mb_query.z.buffer[#bo + 6];
   #r.%B0 := #mb_query.z.buffer[#bo + 7];
   #intreal += DWORD_TO_REAL(#r);
END_FUNCTION

// folder: Library/Modbus/Station blocks/Grundfoss

FUNCTION_BLOCK "Grunnfoss_pump"   // FB14, SCL
{ S7_Optimized_Access := 'TRUE' }
VERSION : 0.1
   VAR_INPUT
      mb_addr : USInt;
      setpoint : Real;   // [%]
   END_VAR
   VAR_OUTPUT
      ProcessFeedback : Real;
      _ : Bool;
      Head : Real;   // bar
      VolumeFlow : Real;   // m3/h
      RelativePerformance : Real;   // %
      Speed : Real;   // rpm
      Frequency : Real;   // Hz
      ActualSetpoint : Real;   // %
      MotorCurrent : Real;   // A
      DCLinkVoltage : Real;   // V
      MotorVoltage : Real;   // V
      Power : Real;   // W
      RemoteFlow : Real;   // m3/h
      InletPressure : Real;   // bar
      RemotePressure : Real;   // bar
      Level : Real;   // m
      PowerElectronicTemp : Real;   // degree C
      MotorTemp : Real;   // degree C
      RemoteTemp : Real;   // degree C
      ElectronicTemp : Real;   // degree C
      PumpLiquidTemp : Real;   // degree C
      BearingTempDE : Real;   // degree C
      BearingTempNDE : Real;   // degree C
      AuxSensorInput : Real;   // %
      SpecificEnergyConsumption : Real;   // Wh/m3
      OperationTime : Real;   // hour
      TotalPoweredTime : Real;   // hour
      Torque : Real;   // Nm
      Energy : Real;   // kWh
      NumberOfStarts : Real;
   END_VAR
   VAR_IN_OUT
      mb_query : "mb_query";
   END_VAR
   VAR
      sb : "mb_station_block_udt";
      read1 : Struct
         status : Struct   // (201)
            x08_AccessModeRemote : Bool;
            x09_On : Bool;
            x10_Fault : Bool;
            x11_Warning : Bool;
            x12_ForcedToLocal : Bool;
            x13_AtMaxSpeed : Bool;
            x14 : Bool;
            x15_AtMinSpeed : Bool;
            x00_LowFlowStop : Bool;
            x01_CopyToLocal : Bool;
            x02_MaxFlowLimitEnabled : Bool;
            x03_ResetAlarmAck : Bool;
            x04_SetpointInfluence : Bool;
            x05_AtMaxPower : Bool;
            x06_Rotation : Bool;
            x07_Direction : Bool;
         END_STRUCT;
         ProcessFeedback : UInt;   // (202) x 0.01
         ControlMode : UInt;   // (203)
         OperationMode : UInt;   // (204)
         AlarmCode : UInt;   // (205)
         WarningCode : UInt;   // (206)
         MonthsToBearingService : Byte;   // (207)
         BearingServiceType : Byte;
         DriveState : UInt;   // (208)
         FeedbackSensorUnit : UInt;   // (209)
         FeedbackSensorMin : UInt;   // (210)
         FeedbackSensorMax : UInt;   // (211)
         NominalFrequency : UInt;   // (212)
         MinFrequency : UInt;   // (213) Minimum frequency in % of nominal frequency
         MaxFrequency : UInt;   // (214) Maximum frequency in % of nominal frequency
         SetpointRangeMin : UInt;   // (215)
         SetpointRangeMax : UInt;   // (216)
         _ : Array[1..4] of UInt;
         FlowEstimationState : UInt;   // (221) 0: within range, 1:below, 2:above
      END_STRUCT;
      read2 : Struct
         Head : UInt;   // (301) 0.001 bar
         VolumeFlow : UInt;   // (302) 0.1 m3/h
         RelativePerformance : UInt;   // (303) 0.01 %
         Speed : UInt;   // (304) rpm
         Frequency : UInt;   // (305) 0.1 Hz
         DigitalInput : Word;   // (306)
         DigitalOutput : Word;   // (307)
         ActualSetpoint : UInt;   // (308) 0.01 %
         MotorCurrent : UInt;   // (309) 0.1 A
         DCLinkVoltage : UInt;   // (310) 0.1 V
         MotorVoltage : UInt;   // (311) 0.1 V
         Power : UDInt;   // (312) W
         RemoteFlow : UInt;   // (314) 0.1 m3/h
         InletPressure : UInt;   // (315) 0.001 bar
         RemotePressure : UInt;   // (316) 0.001 bar
         Level : UInt;   // (317) 0.01 m
         PowerElectronicTemp : UInt;   // (318) 0.01 K
         MotorTemp : UInt;   // (319) 0.01 K
         RemoteTemp : UInt;   // (320) 0.01 K
         ElectronicTemp : UInt;   // (321) 0.01 K
         PumpLiquidTemp : UInt;   // (322) 0.01 K
         BearingTempDE : UInt;   // (323) 0.01 K
         BearingTempNDE : UInt;   // (324) 0.01 K
         AuxSensorInput : UInt;   // (325) 0.01 %
         SpecificEnergyConsumption : UInt;   // (326) Wh/m3
         OperationTime : UDInt;   // (327) hour
         TotalPoweredTime : UDInt;   // (329) hour
         Torque : UInt;   // (331) 0.1 Nm
         Energy : UDInt;   // (332) kWh
         NumberOfStarts : UDInt;   // (334)
      END_STRUCT;
      write : Struct
         cmd : Struct   // (101)
            x08 : Bool;
            x09 : Bool;
            x10 : Bool;
            x11 : Bool;
            x12 : Bool;
            x13 : Bool;
            x14 : Bool;
            x15 : Bool;
            x00_Remote : Bool := true;   // 0=Local
            x01_On : Bool;   // 0=Off
            x02_ResetAlarm : Bool;   // rising edge only
            x03_CopyToLocal : Bool;
            x04_EnableMaxFlowLimit : Bool;
            x05 : Bool;
            x06 : Bool;
            x07 : Bool;
         END_STRUCT;
         ControlMode : UInt;   // (102)
         OperationMode : UInt;   // (103)
         Setpoint : UInt;   // (104)
         Relay : Struct   // (105)
            x08 : Bool;
            x09 : Bool;
            x10 : Bool;
            x11 : Bool;
            x12 : Bool;
            x13 : Bool;
            x14 : Bool;
            x15 : Bool;
            x00_Realy1_inverted : Bool;   // 0: Closed, 1:Open
            x01_Realy2_inverted : Bool;   // 0: Closed, 1:Open
            x02_Realy3_inverted : Bool;   // 0: Closed, 1:Open
            x03_Realy4_inverted : Bool;   // 0: Closed, 1:Open
            x04 : Bool;
            x05 : Bool;
            x06 : Bool;
            x07 : Bool;
            x : Struct
               x08 : Bool;
               x09 : Bool;
               x10 : Bool;
               x11 : Bool;
               x12 : Bool;
               x13 : Bool;
               x14 : Bool;
               x15 : Bool;
               x00 : Bool;
               x01 : Bool;
               x02 : Bool;
               x03 : Bool;
               x04 : Bool;
               x05 : Bool;
               x06 : Bool;
               x07 : Bool;
            END_STRUCT;
            x_1 : Struct
               x08 : Bool;
               x09 : Bool;
               x10 : Bool;
               x11 : Bool;
               x12 : Bool;
               x13 : Bool;
               x14 : Bool;
               x15 : Bool;
               x00 : Bool;
               x01 : Bool;
               x02 : Bool;
               x03 : Bool;
               x04 : Bool;
               x05 : Bool;
               x06 : Bool;
               x07 : Bool;
               x : Struct
                  x08 : Bool;
                  x09 : Bool;
                  x10 : Bool;
                  x11 : Bool;
                  x12 : Bool;
                  x13 : Bool;
                  x14 : Bool;
                  x15 : Bool;
                  x00 : Bool;
                  x01 : Bool;
                  x02 : Bool;
                  x03 : Bool;
                  x04 : Bool;
                  x05 : Bool;
                  x06 : Bool;
                  x07 : Bool;
               END_STRUCT;
            END_STRUCT;
         END_STRUCT;
         SetMaxFlowLimit : UInt;   // (106) 0.01 m3/h
      END_STRUCT;
   END_VAR
BEGIN
   // Grundfoss - Pumps
   // CIM 200 Modbus RTU
   // CIM 500 Modbus TCP

   "mb_station_block_header"(sb := #sb, mb_query := #mb_query);
   #mb_query.mb_addr := #mb_addr;

   #mb_query.mode := #mb_query.c.read.holding_reg;

   #mb_query(data_addr := 201, data_ptr := #read1);
   IF #mb_query.Done THEN
       #ProcessFeedback := UINT_TO_REAL(#read1.ProcessFeedback) / 100;
   END_IF;

   #mb_query(data_addr := 301, data_ptr := #read2);
   IF #mb_query.Done THEN
       #Head := UINT_TO_REAL(#read2.Head) * 0.001;
       #VolumeFlow := UINT_TO_REAL(#read2.VolumeFlow) * 0.1;
       #RelativePerformance := UINT_TO_REAL(#read2.RelativePerformance) * 0.01;
       #Speed := UINT_TO_REAL(#read2.Speed);
       #Frequency := UINT_TO_REAL(#read2.Frequency) * 0.1;
       #ActualSetpoint := UINT_TO_REAL(#read2.ActualSetpoint) * 0.01;
       #MotorCurrent := UINT_TO_REAL(#read2.MotorCurrent) * 0.1;
       #DCLinkVoltage := UINT_TO_REAL(#read2.DCLinkVoltage) * 0.1;
       #MotorVoltage := UINT_TO_REAL(#read2.MotorVoltage) * 0.1;
       #Power := UDINT_TO_REAL(#read2.Power);
       #RemoteFlow := UINT_TO_REAL(#read2.RemoteFlow) * 0.1;
       #InletPressure := UINT_TO_REAL(#read2.InletPressure) * 0.001;
       #RemotePressure := UINT_TO_REAL(#read2.RemotePressure) * 0.001;
       #Level := UINT_TO_REAL(#read2.Level) * 0.01;
       #PowerElectronicTemp := UINT_TO_REAL(#read2.PowerElectronicTemp) * 0.01 - 273.15;
       #MotorTemp := UINT_TO_REAL(#read2.MotorTemp) * 0.01 - 273.15;
       #RemoteTemp := UINT_TO_REAL(#read2.RemoteTemp) * 0.01 - 273.15;
       #ElectronicTemp := UINT_TO_REAL(#read2.ElectronicTemp) * 0.01 - 273.15;
       #PumpLiquidTemp := UINT_TO_REAL(#read2.PumpLiquidTemp) * 0.01 - 273.15;
       #BearingTempDE := UINT_TO_REAL(#read2.BearingTempDE) * 0.01 - 273.15;
       #BearingTempNDE := UINT_TO_REAL(#read2.BearingTempNDE) * 0.01 - 273.15;
       #AuxSensorInput := UINT_TO_REAL(#read2.AuxSensorInput) * 0.01;
       #SpecificEnergyConsumption := UINT_TO_REAL(#read2.SpecificEnergyConsumption);
       #OperationTime := UDINT_TO_REAL(#read2.OperationTime);
       #TotalPoweredTime := UDINT_TO_REAL(#read2.TotalPoweredTime);
       #Torque := UINT_TO_REAL(#read2.Torque) * 0.1;
       #Energy := UDINT_TO_REAL(#read2.Energy);
       #NumberOfStarts := UDINT_TO_REAL(#read2.NumberOfStarts);
   END_IF;


   // Write preparations
   #write.cmd.x01_On := #setpoint <> 0;
   #write.Setpoint := REAL_TO_UINT(#setpoint * 100);

   #mb_query.mode := #mb_query.c.write.holding_reg;
   #mb_query(data_addr := 101, data_ptr := #write);

   "mb_station_block_footer"(sb := #sb, mb_query := #mb_query);

   (*

   #write.ControlMode:
   Some modes are not supported by all E-pumps.
   0: Constant speed
   1: Constant frequency
   3: Constant head
   4: Constant pressure
   5: Constant differential pressure
   6: Proportional pressure
   7: Constant flow
   8: Constant temperature
   10: Constant level
   128: AUTOADAPT
   129: FLOWADAPT (set FLOWLIMIT in register 00106)
   130: Closed-loop sensor.

   #write.OperationMode:
   0: Auto-control (setpoint control according to selected control mode)
   4: OpenLoopMin (running at minimum speed)
   6: OpenLoopMax (running at maximum speed)

   #read.DriveState:
   0: Stopped
   1: Accelerating
   2: Decelerating
   3: Steady state/closed loop
   4: -
   5: Accelerating halt
   6: Decelerating halt
   7: Start on the run (flying cut-in)
   Only MGE motors and CUE drives.

   #read.FeedbackSensorUnit:
   0: bar
   1: mbar
   2: m
   3: kPa
   4: psi
   5: ft
   6: m3/h
   7: m3/s
   8: l/s
   9: gpm
   10: °C
   11: °F
   12: %
   13: K
   14: W

   *)
END_FUNCTION_BLOCK

// folder: Library/Modbus/Station blocks/Honeywell

FUNCTION_BLOCK "Honeywell_UDA2182"   // FB28, SCL
{ S7_Optimized_Access := 'TRUE' }
VERSION : 0.1
   VAR_INPUT
      mb_addr : UInt;
   END_VAR
   VAR_IN_OUT
      mb_query : "mb_query";
   END_VAR
   VAR
      sb : "mb_station_block_udt";
      data : Struct
         pv1 : Array[1..2] of Real;
         temperature : Array[1..2] of Real;
         alarm : Array[1..4] of DWord;
      END_STRUCT;
   END_VAR
BEGIN
   // Honeywell - UDA2182
   // 
   // Web: https://www.honeywellprocess.com/library/support/Public/Documents/70-82-25-126.pdf

   "mb_station_block_header"(sb := #sb, mb_query := #mb_query);
   #mb_query.mb_addr := #mb_addr;

   #mb_query.mode := #mb_query.c.mode.read;
   #mb_query(data_addr := 30001, data_ptr := #data);

   "mb_station_block_footer"(sb := #sb, mb_query := #mb_query);
END_FUNCTION_BLOCK

FUNCTION_BLOCK "Honeywell_variable_frequency_drives"   // FB29, SCL
{ S7_Optimized_Access := 'TRUE' }
VERSION : 0.1
   VAR_INPUT
      mb_addr : UInt := 255;
   END_VAR
   VAR_IN_OUT
      mb_query : "mb_query";
   END_VAR
   VAR
      sb : "mb_station_block_udt";
      read : Struct
         stw : Struct
            x24 : Bool;
            x25 : Bool;
            x26 : Bool;
            x27 : Bool;
            x28 : Bool;
            x29_control_place : Bool := FALSE;
            x30_control_place : Bool := FALSE;
            x31_control_place : Bool := TRUE;
            x16 : Bool;
            x17 : Bool;
            x18 : Bool;
            x19 : Bool;
            x20 : Bool;
            x21 : Bool;
            x22 : Bool;
            x23 : Bool;
            x08 : Bool;
            x09 : Bool;
            x10 : Bool;
            x11 : Bool;
            x12 : Bool;
            x13 : Bool;
            x14 : Bool;
            x15 : Bool;
            x00_Ready : Bool;
            x01_Running : Bool;
            x02_Counterclockwise : Bool;
            x03_Faulted : Bool;
            x04_Alarm : Bool;
            x05_AtReference : Bool;
            x06_ZeroSpeed : Bool;
            x07_FluxReady : Bool;
         END_STRUCT;
         d1_Output_Frequency : DInt;   // 0,01 Hz
         d2_Motor_Speed : DInt;   // 1 rpm
         d3_Motor_Current : DInt;   // 0,1 A
         d4_Motor_Torque : DInt;   // 0,1 %
         d5_Motor_Power : DInt;   // 0,1 %
         d6_Motor_Voltage : DInt;   // 0,1 V
         d7_DC_link_voltage : DInt;   // 1 V
         d8_Active_Fault_Code : DInt;
      END_STRUCT;
      write : Struct
         ctw : Struct
            x08 : Bool;
            x09 : Bool;
            x10 : Bool;
            x11 : Bool;
            x12 : Bool;
            x13 : Bool;
            x14 : Bool;
            x15 : Bool;
            x00 : Bool;
            x01_start : Bool := TRUE;
            x02_Reverse : Bool;
            x03_Reset_faults : Bool;
            x04 : Bool;
            x05 : Bool;
            x06 : Bool;
            x07 : Bool;
         END_STRUCT;
         __ : Word;
         speed_ref : UInt;   // 0â€¦10000 %
      END_STRUCT;
   END_VAR
BEGIN
   // Honeywell - Variable frequency drives
   // 
   // Web: https://customer.honeywell.com/resources/techlit/
   //      TechLitDocuments/62-0000s/62-0351.pdf

   "mb_station_block_header"(sb := #sb, mb_query := #mb_query);
   #mb_query.mb_addr := #mb_addr;

   #mb_query(mode := #mb_query.c.read.holding_reg,
             data_addr := 2151,
             data_ptr := #read);

   #mb_query(mode := #mb_query.c.write.holding_reg,
             data_addr := 2001,
             data_ptr := #write);

   "mb_station_block_footer"(sb := #sb, mb_query := #mb_query);
END_FUNCTION_BLOCK

// folder: Library/Modbus/Station blocks/Krohne

FUNCTION_BLOCK "Krohne_MFC_300"   // FB33, SCL
TITLE = Krohne MFC 300
{ S7_Optimized_Access := 'TRUE' }
AUTHOR : OlaBjornli
FAMILY : modbus
VERSION : 0.1
// Coriolise flow meter
   VAR_INPUT
      mb_addr : UInt;
   END_VAR
   VAR_OUTPUT
      Temperature : Real;   // [degree C]
   END_VAR
   VAR_IN_OUT
      mb_query : "mb_query";
   END_VAR
   VAR
      sb : "mb_station_block_udt";
      read1 : Struct
         "Flow Velocity" : Real;   // [m/s]
         "Volume Flow" : Real;   // [m3/s]
         "Mass Flow" : Real;   // [kg/s]
         Temperature : Real := 273.15;   // [K]
         Density : Real;   // [kg/m3]
         Concentration_1 : Real;
         Concentration_2_or_Diagnosis_3 : Real;
         Concentration_Flow_1 : Real;
         Concentration_Flow_2 : Real;
         Diagnosis_1 : Real;
         Diagnosis_2 : Real;
         Display_Channel_1 : Real;
         Display_Channel_2 : Real;
         Operating_time : Real;   // [s]
      END_STRUCT;
      write1_settings : Struct
         Counter_1_Function : UInt;
         Counter_1_Measurement : UInt;
         Counter_2_Function : UInt;
         Counter_2_Measurement : UInt;
         Counter_3_Function : UInt;
         Counter_3_Measurement : UInt;
      END_STRUCT;
      exec_write : Bool;
   END_VAR
BEGIN
   // Krohne - MFC 300 
   // Flowmeter
   // 
   // Web: http://cdn.krohne.com/dlc/AD_MFC300_Modbus_en_091124_4000744801_R01.pdf
   //
   // #settings :
   //    Counter Function:
   //       1 = Sum Counter
   //       2 = + Counter
   //       3 = - Counter
   //       0 = Off
   //    Counter Measurement:
   //       21 = Volume Flow [m3]
   //       22 = Mass Flow [kg]
   //       27 = Concentration Flow 1
   //       28 = Concentration Flow 2

   "mb_station_block_header"(sb := #sb, mb_query := #mb_query);
   #mb_query.mb_addr := #mb_addr;

   #mb_query(mode := #mb_query.c.mode.read,
             data_addr := 30001, // 30000 + 1 (error in datasheet)
             data_ptr := #read1);
   #Temperature := #read1.Temperature - 273.15;

   // The write query isn't executing continuously in case that will damage eeprom
   IF #exec_write THEN
       #mb_query(mode := #mb_query.c.mode.write,
                 data_addr := 40001, // 40000 + 1,
                 data_ptr := #write1_settings);
       #exec_write := NOT #mb_query.Done;
   END_IF;

   "mb_station_block_footer"(sb := #sb, mb_query := #mb_query);
END_FUNCTION_BLOCK

FUNCTION_BLOCK "Krohne_Optisonic"   // FB34, SCL
{ S7_Optimized_Access := 'TRUE' }
VERSION : 0.1
   VAR_INPUT
      mb_addr : UInt;
   END_VAR
   VAR_IN_OUT
      mb_query : "mb_query";
   END_VAR
   VAR
      sb : "mb_station_block_udt";
      data : Struct
         "Temperature process value" : Real;
         "Dynamic Viscosity at Process conditions" : Real;
         "Density Process" : Real;
         "Flow Process" : Real;
         "Velocity Process" : Real;
         "Speed of Sound" : Real;
      END_STRUCT;
   END_VAR
BEGIN
   // Krohne - Optisonic V6
   // 

   "mb_station_block_header"(sb := #sb,
                             mb_query := #mb_query);
   #mb_query.mb_addr := #mb_addr;

   #mb_query.mode := #mb_query.c.read.holding_reg;
   #mb_query(data_addr := 7050,
             data_ptr := #data);

   "mb_station_block_footer"(sb := #sb,
                             mb_query := #mb_query);
END_FUNCTION_BLOCK

// folder: Library/Modbus/Station blocks/Mettler

FUNCTION_BLOCK "mettler_toledo_IND560_loadTargetValue"   // FB87, SCL
{ S7_Optimized_Access := 'TRUE' }
VERSION : 0.1
   VAR_INPUT
      iValue : Real;
   END_VAR
   VAR_OUTPUT
      qDone : Bool;
   END_VAR
   VAR_IN_OUT
      "M" : "mettlerToledoInd560Udt";
      sb : "mb_station_block_udt";
   END_VAR
   VAR
      state : Int;
      old_value : Real;
      slot : USInt;
   END_VAR
   VAR CONSTANT
      NONE_AVAILABLE : USInt := 0;
   END_VAR
BEGIN
   // Load target value, for scale 1. Page 143, table B-6

   CASE #state OF

       0:  // Waiting for start.
           #qDone := false;
           #state +=
           BOOL_TO_INT(#old_value <> #iValue);

       1:  // Wait for available msg. slot
           #slot := "reqMsgSlot"(#"M".occupiedMsgSlots);
           #state += BOOL_TO_INT(#slot <> #NONE_AVAILABLE);

       2:  // #1 PLC loads floating point value first
           #"M".writeMsgSlot[#slot].cmd := 0;
           #"M".writeMsgSlot[#slot].data := #iValue;
           #state += 1;
       3:
           #state += BOOL_TO_INT(#"M".queryDone.write);

       4:  // #2 PLC sends command to set target 1 cutoff value 
           #"M".writeMsgSlot[#slot].cmd := 110;
           #state += 1;
       5:
           #state += BOOL_TO_INT(#"M".queryDone.write);

       6:  // #3 IND560 terminal sees new command, loads the value into the target
           //    and ends a return message to indicate the new target value.
           #state +=
           BOOL_TO_INT(#"M".queryDone.read
                       AND #"M".run.cmdAck[#slot] = 1
                       AND #"M".run.PF[#slot] = 13
                       AND #"M".readMsgSlot[#slot].data = #"M".writeMsgSlot[#slot].data);

       7:  // #4  PLC instructs IND560 terminal to start â€œusingâ€ new target value
           #"M".writeMsgSlot[#slot].cmd := 114;
           #state += 1;
       8:
           #state += BOOL_TO_INT(#"M".queryDone.write);

       9:  // #5 IND560 terminal sees new command
           #"M".writeMsgSlot[#slot].cmd := 0;

           #state +=
           BOOL_TO_INT(#"M".queryDone.read
                       AND #"M".run.cmdAck[#slot] = 2
                       AND #"M".run.PF[#slot] = 30
                       AND #"M".readMsgSlot[#slot].data = 0);

       ELSE: // Back to start.
           #"M".occupiedMsgSlots[#slot] := false; // Release msg. slot.
           #state := 0;
           #qDone := true;
           // The start signal should need to be set back false before next
           // exec. else the sequence will start over.
   END_CASE;
   #old_value := #iValue;

   // 
   IF #sb.out.error_comm THEN
       #state := 0;
       IF #slot <> #NONE_AVAILABLE THEN
           #"M".writeMsgSlot[#slot].cmd := 0;
           "releaseMsgSlot"(slot := #slot,
                            mem := #"M".occupiedMsgSlots);
       END_IF;
   END_IF;
END_FUNCTION_BLOCK

FUNCTION_BLOCK "mettler_toledo_IND560"   // FB88, SCL
{ S7_Optimized_Access := 'TRUE' }
VERSION : 0.1
   VAR_IN_OUT
      mb_query : "mb_query";
   END_VAR
   VAR
      mb_addr : UInt := 255;
      sb : "mb_station_block_udt";
      "M" : "mettlerToledoInd560Udt";   // Shared data
      loadTargetValue : "mettler_toledo_IND560_loadTargetValue";
      s : USInt;
   END_VAR
   VAR_TEMP
      c : Int;
   END_VAR
BEGIN
   // Mettler Toledo IND560 - Weighing Terminal

   // WARNING: This SB is just a draft and the block probably include errors !!

   // Necessary settings: ()
   // PLC -> Eth/IP - Modbus TCP -> IP-address
   // PLC -> Eth/IP - Modbus TCP -> Subnet-mask
   // PLC -> Data Format -> Byte order : standard
   // PLC -> Data Format -> Format     : Floating Point 

